LIN {X 0,Y 544.35,Z 282.985,A -85,B 0,C 180,E1 26412.669,E2 26412.669} C_VEL
LIN {X 0,Y 544.407,Z 282.987,A -85,B 0,C 180,E1 26409.453,E2 26409.453} C_VEL
LIN {X 0,Y 544.348,Z 282.987,A -85,B 0,C 180,E1 26406.128,E2 26406.128} C_VEL
LIN {X 0,Y 544.355,Z 282.985,A -85,B 0,C 180,E1 26402.683,E2 26402.683} C_VEL
LIN {X 0,Y 544.403,Z 282.989,A -85,B 0,C 180,E1 26399.482,E2 26399.482} C_VEL
LIN {X 0,Y 544.346,Z 282.986,A -85,B 0,C 180,E1 26396.273,E2 26396.273} C_VEL
LIN {X 0,Y 544.393,Z 282.983,A -85,B 0,C 180,E1 26393.029,E2 26393.029} C_VEL
LIN {X 0,Y 544.372,Z 282.987,A -85,B 0,C 180,E1 26389.751,E2 26389.751} C_VEL
LIN {X 0,Y 544.351,Z 282.985,A -85,B 0,C 180,E1 26386.43,E2 26386.43} C_VEL
LIN {X 0,Y 544.405,Z 282.984,A -85,B 0,C 180,E1 26383.163,E2 26383.163} C_VEL
LIN {X 0,Y 544.358,Z 282.987,A -85,B 0,C 180,E1 26379.941,E2 26379.941} C_VEL
LIN {X 0,Y 544.356,Z 282.984,A -85,B 0,C 180,E1 26376.463,E2 26376.463} C_VEL
LIN {X 0,Y 544.404,Z 282.984,A -85,B 0,C 180,E1 26373.158,E2 26373.158} C_VEL
LIN {X 0,Y 544.36,Z 282.986,A -85,B 0,C 180,E1 26369.894,E2 26369.894} C_VEL
LIN {X 0,Y 544.358,Z 282.984,A -85,B 0,C 180,E1 26366.419,E2 26366.419} C_VEL
LIN {X 0,Y 544.407,Z 282.984,A -85,B 0,C 180,E1 26363.143,E2 26363.143} C_VEL
LIN {X 0,Y 544.363,Z 282.986,A -85,B 0,C 180,E1 26359.843,E2 26359.843} C_VEL
LIN {X 0,Y 544.361,Z 282.984,A -85,B 0,C 180,E1 26356.401,E2 26356.401} C_VEL
LIN {X 0,Y 544.406,Z 282.984,A -85,B 0,C 180,E1 26353.102,E2 26353.102} C_VEL
LIN {X 0,Y 544.366,Z 282.986,A -85,B 0,C 180,E1 26349.799,E2 26349.799} C_VEL
LIN {X 0,Y 544.365,Z 282.983,A -85,B 0,C 180,E1 26346.395,E2 26346.395} C_VEL
LIN {X 0,Y 544.406,Z 282.985,A -85,B 0,C 180,E1 26343.14,E2 26343.14} C_VEL
LIN {X 0,Y 544.362,Z 282.985,A -85,B 0,C 180,E1 26339.89,E2 26339.89} C_VEL
LIN {X 0,Y 544.374,Z 282.982,A -85,B 0,C 180,E1 26336.493,E2 26336.493} C_VEL
LIN {X 0,Y 544.405,Z 282.986,A -85,B 0,C 180,E1 26333.199,E2 26333.199} C_VEL
LIN {X 0,Y 544.361,Z 282.985,A -85,B 0,C 180,E1 26329.986,E2 26329.986} C_VEL
LIN {X 0,Y 544.389,Z 282.981,A -85,B 0,C 180,E1 26326.613,E2 26326.613} C_VEL
LIN {X 0,Y 544.401,Z 282.989,A -85,B 0,C 180,E1 26323.237,E2 26323.237} C_VEL
LIN {X 0,Y 544.364,Z 282.985,A -85,B 0,C 180,E1 26320.002,E2 26320.002} C_VEL
LIN {X 0,Y 544.398,Z 282.982,A -85,B 0,C 180,E1 26316.646,E2 26316.646} C_VEL
LIN {X 0,Y 544.397,Z 282.989,A -85,B 0,C 180,E1 26313.306,E2 26313.306} C_VEL
LIN {X 0,Y 544.365,Z 282.988,A -85,B 0,C 180,E1 26309.971,E2 26309.971} C_VEL
LIN {X 0,Y 544.436,Z 283.218,A -85,B 0,C 180,E1 26308.729,E2 26308.729} C_VEL
LIN {X 0,Y 547.156,Z 294.377,A -85,B 0,C 180,E1 26307.24,E2 26307.24} C_VEL
LIN {X 0,Y 546.527,Z 321.838,A -85,B 0,C 180,E1 26304.018,E2 26304.018} C_VEL
LIN {X 0,Y 545.809,Z 351.894,A -85,B 0,C 180,E1 26300.535,E2 26300.535} C_VEL
LIN {X 0,Y 545.233,Z 382.464,A -85,B 0,C 180,E1 26297.06,E2 26297.06} C_VEL
LIN {X 0,Y 544.899,Z 404.895,A -85,B 0,C 180,E1 26294.573,E2 26294.573} C_VEL
LIN {X 0,Y 545.732,Z 413.339,A -85,B 0,C 180,E1 26294.433,E2 26294.433} C_VEL
LIN {X 0,Y 545.362,Z 516.208,A -85,B 0,C 180,E1 26293.038,E2 26293.038} C_VEL
LIN {X 0,Y 545.216,Z 531.178,A -85,B 0,C 180,E1 26292.642,E2 26292.642} C_VEL
LIN {X 0,Y 544.986,Z 546.217,A -85,B 0,C 180,E1 26292.017,E2 26292.017} C_VEL
LIN {X 0,Y 544.757,Z 559.301,A -85,B 0,C 180,E1 26291.265,E2 26291.265} C_VEL
LIN {X 0,Y 544.54,Z 571.401,A -85,B 0,C 180,E1 26290.365,E2 26290.365} C_VEL
LIN {X 0,Y 544.321,Z 583.569,A -85,B 0,C 180,E1 26289.194,E2 26289.194} C_VEL
LIN {X 0,Y 544.146,Z 593.806,A -85,B 0,C 180,E1 26287.92,E2 26287.92} C_VEL
LIN {X 0,Y 544.035,Z 601.785,A -85,B 0,C 180,E1 26286.647,E2 26286.647} C_VEL
LIN {X 0,Y 543.96,Z 608.864,A -85,B 0,C 180,E1 26285.166,E2 26285.166} C_VEL
LIN {X 0,Y 543.928,Z 614.181,A -85,B 0,C 180,E1 26283.582,E2 26283.582} C_VEL
LIN {X 0,Y 543.917,Z 617.464,A -85,B 0,C 180,E1 26282,E2 26282} C_VEL
LIN {X 0,Y 543.918,Z 618.907,A -85,B 0,C 180,E1 26280.42,E2 26280.42} C_VEL
LIN {X 0,Y 543.915,Z 618.544,A -85,B 0,C 180,E1 26278.84,E2 26278.84} C_VEL
LIN {X 0,Y 543.919,Z 616.339,A -85,B 0,C 180,E1 26277.259,E2 26277.259} C_VEL
LIN {X 0,Y 543.935,Z 612.587,A -85,B 0,C 180,E1 26275.782,E2 26275.782} C_VEL
LIN {X 0,Y 543.983,Z 606.506,A -85,B 0,C 180,E1 26274.197,E2 26274.197} C_VEL
LIN {X 0,Y 544.068,Z 599.221,A -85,B 0,C 180,E1 26272.82,E2 26272.82} C_VEL
LIN {X 0,Y 544.2,Z 590.528,A -85,B 0,C 180,E1 26271.546,E2 26271.546} C_VEL
LIN {X 0,Y 544.389,Z 579.839,A -85,B 0,C 180,E1 26270.324,E2 26270.324} C_VEL
LIN {X 0,Y 544.589,Z 567.853,A -85,B 0,C 180,E1 26269.259,E2 26269.259} C_VEL
LIN {X 0,Y 544.837,Z 555.527,A -85,B 0,C 180,E1 26268.406,E2 26268.406} C_VEL
LIN {X 0,Y 545.075,Z 541.334,A -85,B 0,C 180,E1 26267.659,E2 26267.659} C_VEL
LIN {X 0,Y 545.291,Z 525.913,A -85,B 0,C 180,E1 26267.099,E2 26267.099} C_VEL
LIN {X 0,Y 545.406,Z 510.362,A -85,B 0,C 180,E1 26266.767,E2 26266.767} C_VEL
LIN {X 0,Y 545.638,Z 409.282,A -85,B 0,C 180,E1 26265.372,E2 26265.372} C_VEL
LIN {X 0,Y 544.953,Z 404.69,A -85,B 0,C 180,E1 26265.278,E2 26265.278} C_VEL
LIN {X 0,Y 545.578,Z 374.772,A -85,B 0,C 180,E1 26261.846,E2 26261.846} C_VEL
LIN {X 0,Y 546.318,Z 345.052,A -85,B 0,C 180,E1 26258.394,E2 26258.394} C_VEL
LIN {X 0,Y 547.209,Z 316.527,A -85,B 0,C 180,E1 26255.033,E2 26255.033} C_VEL
LIN {X 0,Y 547.803,Z 295.13,A -85,B 0,C 180,E1 26252.444,E2 26252.444} C_VEL
LIN {X 0,Y 544.407,Z 282.987,A -85,B 0,C 180,E1 26250.634,E2 26250.634} C_VEL
LIN {X 0,Y 544.383,Z 282.99,A -85,B 0,C 180,E1 26247.268,E2 26247.268} C_VEL
LIN {X 0,Y 544.383,Z 282.986,A -85,B 0,C 180,E1 26243.872,E2 26243.872} C_VEL
LIN {X 0,Y 544.393,Z 282.984,A -85,B 0,C 180,E1 26240.544,E2 26240.544} C_VEL
LIN {X 0,Y 544.39,Z 282.988,A -85,B 0,C 180,E1 26237.125,E2 26237.125} C_VEL
LIN {X 0,Y 544.402,Z 282.987,A -85,B 0,C 180,E1 26233.797,E2 26233.797} C_VEL
LIN {X 0,Y 544.387,Z 282.985,A -85,B 0,C 180,E1 26230.418,E2 26230.418} C_VEL
LIN {X 0,Y 544.353,Z 282.99,A -85,B 0,C 180,E1 26227.047,E2 26227.047} C_VEL
LIN {X 0,Y 544.384,Z 282.991,A -85,B 0,C 180,E1 26223.816,E2 26223.816} C_VEL
LIN {X 0,Y 544.345,Z 283.033,A -85,B 0,C 180,E1 26222.92,E2 26222.92} C_VEL
LIN {X 0,Y 549.395,Z 298.474,A -85,B 0,C 180,E1 26221.305,E2 26221.305} C_VEL
LIN {X 0,Y 548.406,Z 338.599,A -85,B 0,C 180,E1 26218.283,E2 26218.283} C_VEL
LIN {X 0,Y 547.611,Z 384.589,A -85,B 0,C 180,E1 26215.005,E2 26215.005} C_VEL
LIN {X 0,Y 547.643,Z 387.567,A -85,B 0,C 180,E1 26214.823,E2 26214.823} C_VEL
LIN {X 0,Y 548.835,Z 396.99,A -85,B 0,C 180,E1 26214.653,E2 26214.653} C_VEL
LIN {X 0,Y 548.051,Z 589.9,A -85,B 0,C 180,E1 26212.072,E2 26212.072} C_VEL
LIN {X 0,Y 547.776,Z 609.321,A -85,B 0,C 180,E1 26211.669,E2 26211.669} C_VEL
LIN {X 0,Y 547.427,Z 627.661,A -85,B 0,C 180,E1 26211.09,E2 26211.09} C_VEL
LIN {X 0,Y 546.99,Z 645.573,A -85,B 0,C 180,E1 26210.323,E2 26210.323} C_VEL
LIN {X 0,Y 546.512,Z 662.304,A -85,B 0,C 180,E1 26209.409,E2 26209.409} C_VEL
LIN {X 0,Y 546.011,Z 678.751,A -85,B 0,C 180,E1 26208.296,E2 26208.296} C_VEL
LIN {X 0,Y 545.512,Z 694.468,A -85,B 0,C 180,E1 26206.999,E2 26206.999} C_VEL
LIN {X 0,Y 545.083,Z 708.249,A -85,B 0,C 180,E1 26205.63,E2 26205.63} C_VEL
LIN {X 0,Y 544.714,Z 720.88,A -85,B 0,C 180,E1 26204.131,E2 26204.131} C_VEL
LIN {X 0,Y 544.42,Z 732.249,A -85,B 0,C 180,E1 26202.517,E2 26202.517} C_VEL
LIN {X 0,Y 544.199,Z 742.233,A -85,B 0,C 180,E1 26200.802,E2 26200.802} C_VEL
LIN {X 0,Y 544.052,Z 750.798,A -85,B 0,C 180,E1 26198.988,E2 26198.988} C_VEL
LIN {X 0,Y 543.974,Z 757.523,A -85,B 0,C 180,E1 26197.181,E2 26197.181} C_VEL
LIN {X 0,Y 543.932,Z 762.857,A -85,B 0,C 180,E1 26195.274,E2 26195.274} C_VEL
LIN {X 0,Y 543.911,Z 766.48,A -85,B 0,C 180,E1 26193.373,E2 26193.373} C_VEL
LIN {X 0,Y 543.912,Z 768.551,A -85,B 0,C 180,E1 26191.37,E2 26191.37} C_VEL
LIN {X 0,Y 543.913,Z 768.872,A -85,B 0,C 180,E1 26189.369,E2 26189.369} C_VEL
LIN {X 0,Y 543.911,Z 767.453,A -85,B 0,C 180,E1 26187.367,E2 26187.367} C_VEL
LIN {X 0,Y 543.92,Z 764.466,A -85,B 0,C 180,E1 26185.467,E2 26185.467} C_VEL
LIN {X 0,Y 543.946,Z 759.811,A -85,B 0,C 180,E1 26183.563,E2 26183.563} C_VEL
LIN {X 0,Y 544.019,Z 753.373,A -85,B 0,C 180,E1 26181.652,E2 26181.652} C_VEL
LIN {X 0,Y 544.141,Z 745.484,A -85,B 0,C 180,E1 26179.841,E2 26179.841} C_VEL
LIN {X 0,Y 544.342,Z 735.601,A -85,B 0,C 180,E1 26178.021,E2 26178.021} C_VEL
LIN {X 0,Y 544.624,Z 724.151,A -85,B 0,C 180,E1 26176.302,E2 26176.302} C_VEL
LIN {X 0,Y 544.998,Z 711.102,A -85,B 0,C 180,E1 26174.682,E2 26174.682} C_VEL
LIN {X 0,Y 545.442,Z 696.892,A -85,B 0,C 180,E1 26173.22,E2 26173.22} C_VEL
LIN {X 0,Y 545.932,Z 681.441,A -85,B 0,C 180,E1 26171.904,E2 26171.904} C_VEL
LIN {X 0,Y 546.426,Z 665.205,A -85,B 0,C 180,E1 26170.768,E2 26170.768} C_VEL
LIN {X 0,Y 546.924,Z 647.857,A -85,B 0,C 180,E1 26169.787,E2 26169.787} C_VEL
LIN {X 0,Y 547.377,Z 629.851,A -85,B 0,C 180,E1 26168.991,E2 26168.991} C_VEL
LIN {X 0,Y 547.749,Z 611.346,A -85,B 0,C 180,E1 26168.385,E2 26168.385} C_VEL
LIN {X 0,Y 548.034,Z 592.5,A -85,B 0,C 180,E1 26167.97,E2 26167.97} C_VEL
LIN {X 0,Y 548.83,Z 394.706,A -85,B 0,C 180,E1 26165.294,E2 26165.294} C_VEL
LIN {X 0,Y 547.652,Z 386.629,A -85,B 0,C 180,E1 26165.114,E2 26165.114} C_VEL
LIN {X 0,Y 548.643,Z 339.725,A -85,B 0,C 180,E1 26161.718,E2 26161.718} C_VEL
LIN {X 0,Y 549.499,Z 299.011,A -85,B 0,C 180,E1 26158.703,E2 26158.703} C_VEL
LIN {X 0,Y 547.135,Z 291.4,A -85,B 0,C 180,E1 26157.988,E2 26157.988} C_VEL
LIN {X 0,Y 544.332,Z 282.995,A -85,B 0,C 180,E1 26157.132,E2 26157.132} C_VEL
LIN {X 0,Y 544.372,Z 282.991,A -85,B 0,C 180,E1 26154.004,E2 26154.004} C_VEL
LIN {X 0,Y 544.32,Z 282.991,A -85,B 0,C 180,E1 26150.811,E2 26150.811} C_VEL
LIN {X 0,Y 544.377,Z 282.99,A -85,B 0,C 180,E1 26147.592,E2 26147.592} C_VEL
LIN {X 0,Y 544.329,Z 282.99,A -85,B 0,C 180,E1 26144.396,E2 26144.396} C_VEL
LIN {X 0,Y 544.325,Z 282.99,A -85,B 0,C 180,E1 26140.979,E2 26140.979} C_VEL
LIN {X 0,Y 544.385,Z 282.989,A -85,B 0,C 180,E1 26137.838,E2 26137.838} C_VEL
LIN {X 0,Y 544.323,Z 282.989,A -85,B 0,C 180,E1 26134.584,E2 26134.584} C_VEL
LIN {X 0,Y 544.354,Z 282.988,A -85,B 0,C 180,E1 26131.32,E2 26131.32} C_VEL
LIN {X 0,Y 544.336,Z 282.989,A -85,B 0,C 180,E1 26128.289,E2 26128.289} C_VEL
LIN {X 0,Y 544.328,Z 282.988,A -85,B 0,C 180,E1 26124.876,E2 26124.876} C_VEL
LIN {X 0,Y 544.396,Z 282.989,A -85,B 0,C 180,E1 26121.665,E2 26121.665} C_VEL
LIN {X 0,Y 544.33,Z 282.988,A -85,B 0,C 180,E1 26118.419,E2 26118.419} C_VEL
LIN {X 0,Y 544.336,Z 282.988,A -85,B 0,C 180,E1 26114.948,E2 26114.948} C_VEL
LIN {X 0,Y 544.386,Z 282.989,A -85,B 0,C 180,E1 26111.765,E2 26111.765} C_VEL
LIN {X 0,Y 544.328,Z 282.988,A -85,B 0,C 180,E1 26108.558,E2 26108.558} C_VEL
LIN {X 0,Y 544.381,Z 282.987,A -85,B 0,C 180,E1 26105.376,E2 26105.376} C_VEL
LIN {X 0,Y 544.341,Z 282.988,A -85,B 0,C 180,E1 26102.212,E2 26102.212} C_VEL
LIN {X 0,Y 544.338,Z 282.987,A -85,B 0,C 180,E1 26098.844,E2 26098.844} C_VEL
LIN {X 0,Y 544.397,Z 282.989,A -85,B 0,C 180,E1 26095.577,E2 26095.577} C_VEL
LIN {X 0,Y 544.333,Z 282.988,A -85,B 0,C 180,E1 26092.402,E2 26092.402} C_VEL
LIN {X 0,Y 544.361,Z 282.986,A -85,B 0,C 180,E1 26089.097,E2 26089.097} C_VEL
LIN {X 0,Y 544.359,Z 282.988,A -85,B 0,C 180,E1 26085.971,E2 26085.971} C_VEL
LIN {X 0,Y 544.339,Z 282.986,A -85,B 0,C 180,E1 26082.69,E2 26082.69} C_VEL
LIN {X 0,Y 544.402,Z 282.987,A -85,B 0,C 180,E1 26079.466,E2 26079.466} C_VEL
LIN {X 0,Y 544.339,Z 282.987,A -85,B 0,C 180,E1 26076.282,E2 26076.282} C_VEL
LIN {X 0,Y 544.355,Z 282.986,A -85,B 0,C 180,E1 26072.904,E2 26072.904} C_VEL
LIN {X 0,Y 544.385,Z 282.989,A -85,B 0,C 180,E1 26069.68,E2 26069.68} C_VEL
LIN {X 0,Y 544.383,Z 282.985,A -85,B 0,C 180,E1 26069.164,E2 26069.164} C_VEL
LIN {X 0,Y 543.331,Z 283.113,A -85,B 0,C 180,E1 26068.354,E2 26068.354} C_VEL
LIN {X 0,Y 536.958,Z 283.922,A -85,B 0,C 180,E1 26066.077,E2 26066.077} C_VEL
LIN {X 0,Y 536.46,Z 283.977,A -85,B 0,C 180,E1 26065.485,E2 26065.485} C_VEL
LIN {X 0,Y 536.406,Z 283.976,A -85,B 0,C 180,E1 26062.178,E2 26062.178} C_VEL
LIN {X 0,Y 536.41,Z 283.974,A -85,B 0,C 180,E1 26058.692,E2 26058.692} C_VEL
LIN {X 0,Y 536.464,Z 283.975,A -85,B 0,C 180,E1 26055.363,E2 26055.363} C_VEL
LIN {X 0,Y 536.41,Z 283.976,A -85,B 0,C 180,E1 26052.113,E2 26052.113} C_VEL
LIN {X 0,Y 536.412,Z 283.974,A -85,B 0,C 180,E1 26048.639,E2 26048.639} C_VEL
LIN {X 0,Y 536.462,Z 283.976,A -85,B 0,C 180,E1 26045.424,E2 26045.424} C_VEL
LIN {X 0,Y 536.408,Z 283.975,A -85,B 0,C 180,E1 26042.199,E2 26042.199} C_VEL
LIN {X 0,Y 536.43,Z 283.973,A -85,B 0,C 180,E1 26038.837,E2 26038.837} C_VEL
LIN {X 0,Y 536.451,Z 283.977,A -85,B 0,C 180,E1 26035.571,E2 26035.571} C_VEL
LIN {X 0,Y 536.41,Z 283.975,A -85,B 0,C 180,E1 26032.233,E2 26032.233} C_VEL
LIN {X 0,Y 536.444,Z 283.972,A -85,B 0,C 180,E1 26028.923,E2 26028.923} C_VEL
LIN {X 0,Y 536.451,Z 283.977,A -85,B 0,C 180,E1 26025.568,E2 26025.568} C_VEL
LIN {X 0,Y 536.411,Z 283.974,A -85,B 0,C 180,E1 26022.268,E2 26022.268} C_VEL
LIN {X 0,Y 536.453,Z 283.972,A -85,B 0,C 180,E1 26018.966,E2 26018.966} C_VEL
LIN {X 0,Y 536.439,Z 283.976,A -85,B 0,C 180,E1 26015.668,E2 26015.668} C_VEL
LIN {X 0,Y 536.416,Z 283.973,A -85,B 0,C 180,E1 26012.349,E2 26012.349} C_VEL
LIN {X 0,Y 536.463,Z 283.972,A -85,B 0,C 180,E1 26009.038,E2 26009.038} C_VEL
LIN {X 0,Y 536.437,Z 283.976,A -85,B 0,C 180,E1 26005.659,E2 26005.659} C_VEL
LIN {X 0,Y 536.417,Z 283.973,A -85,B 0,C 180,E1 26002.287,E2 26002.287} C_VEL
LIN {X 0,Y 536.46,Z 283.971,A -85,B 0,C 180,E1 25998.931,E2 25998.931} C_VEL
LIN {X 0,Y 536.446,Z 283.977,A -85,B 0,C 180,E1 25995.536,E2 25995.536} C_VEL
LIN {X 0,Y 536.419,Z 283.973,A -85,B 0,C 180,E1 25992.2,E2 25992.2} C_VEL
LIN {X 0,Y 536.466,Z 283.97,A -85,B 0,C 180,E1 25988.917,E2 25988.917} C_VEL
LIN {X 0,Y 536.443,Z 283.976,A -85,B 0,C 180,E1 25985.557,E2 25985.557} C_VEL
LIN {X 0,Y 536.423,Z 283.973,A -85,B 0,C 180,E1 25982.225,E2 25982.225} C_VEL
LIN {X 0,Y 536.467,Z 283.971,A -85,B 0,C 180,E1 25978.917,E2 25978.917} C_VEL
LIN {X 0,Y 536.439,Z 283.976,A -85,B 0,C 180,E1 25975.614,E2 25975.614} C_VEL
LIN {X 0,Y 536.425,Z 283.973,A -85,B 0,C 180,E1 25972.176,E2 25972.176} C_VEL
LIN {X 0,Y 536.467,Z 283.97,A -85,B 0,C 180,E1 25968.844,E2 25968.844} C_VEL
LIN {X 0,Y 536.454,Z 283.977,A -85,B 0,C 180,E1 25965.393,E2 25965.393} C_VEL
LIN {X 0,Y 536.425,Z 283.973,A -85,B 0,C 180,E1 25961.998,E2 25961.998} C_VEL
LIN {X 0,Y 536.458,Z 283.971,A -85,B 0,C 180,E1 25958.634,E2 25958.634} C_VEL
LIN {X 0,Y 536.459,Z 283.977,A -85,B 0,C 180,E1 25955.278,E2 25955.278} C_VEL
LIN {X 0,Y 536.425,Z 283.974,A -85,B 0,C 180,E1 25951.959,E2 25951.959} C_VEL
LIN {X 0,Y 536.486,Z 284.117,A -85,B 0,C 180,E1 25949.086,E2 25949.086} C_VEL
LIN {X 0,Y 539.574,Z 296.864,A -85,B 0,C 180,E1 25947.356,E2 25947.356} C_VEL
LIN {X 0,Y 538.85,Z 324.871,A -85,B 0,C 180,E1 25944.033,E2 25944.033} C_VEL
LIN {X 0,Y 538.045,Z 354.443,A -85,B 0,C 180,E1 25940.56,E2 25940.56} C_VEL
LIN {X 0,Y 537.397,Z 384.529,A -85,B 0,C 180,E1 25937.094,E2 25937.094} C_VEL
LIN {X 0,Y 537.089,Z 404.785,A -85,B 0,C 180,E1 25934.837,E2 25934.837} C_VEL
LIN {X 0,Y 538.058,Z 413.957,A -85,B 0,C 180,E1 25934.666,E2 25934.666} C_VEL
LIN {X 0,Y 537.621,Z 515.567,A -85,B 0,C 180,E1 25933.263,E2 25933.263} C_VEL
LIN {X 0,Y 537.452,Z 531.399,A -85,B 0,C 180,E1 25932.847,E2 25932.847} C_VEL
LIN {X 0,Y 537.214,Z 545.837,A -85,B 0,C 180,E1 25932.248,E2 25932.248} C_VEL
LIN {X 0,Y 536.96,Z 559.078,A -85,B 0,C 180,E1 25931.491,E2 25931.491} C_VEL
LIN {X 0,Y 536.7,Z 571.358,A -85,B 0,C 180,E1 25930.572,E2 25930.572} C_VEL
LIN {X 0,Y 536.443,Z 583.028,A -85,B 0,C 180,E1 25929.439,E2 25929.439} C_VEL
LIN {X 0,Y 536.237,Z 592.62,A -85,B 0,C 180,E1 25928.253,E2 25928.253} C_VEL
LIN {X 0,Y 536.075,Z 601.425,A -85,B 0,C 180,E1 25926.854,E2 25926.854} C_VEL
LIN {X 0,Y 535.976,Z 608.485,A -85,B 0,C 180,E1 25925.35,E2 25925.35} C_VEL
LIN {X 0,Y 535.931,Z 613.881,A -85,B 0,C 180,E1 25923.742,E2 25923.742} C_VEL
LIN {X 0,Y 535.918,Z 617.146,A -85,B 0,C 180,E1 25922.244,E2 25922.244} C_VEL
LIN {X 0,Y 535.918,Z 618.828,A -85,B 0,C 180,E1 25920.64,E2 25920.64} C_VEL
LIN {X 0,Y 535.915,Z 618.68,A -85,B 0,C 180,E1 25919.036,E2 25919.036} C_VEL
LIN {X 0,Y 535.919,Z 616.751,A -85,B 0,C 180,E1 25917.432,E2 25917.432} C_VEL
LIN {X 0,Y 535.936,Z 612.913,A -85,B 0,C 180,E1 25915.826,E2 25915.826} C_VEL
LIN {X 0,Y 535.995,Z 607.122,A -85,B 0,C 180,E1 25914.217,E2 25914.217} C_VEL
LIN {X 0,Y 536.106,Z 600.193,A -85,B 0,C 180,E1 25912.82,E2 25912.82} C_VEL
LIN {X 0,Y 536.276,Z 591.881,A -85,B 0,C 180,E1 25911.529,E2 25911.529} C_VEL
LIN {X 0,Y 536.509,Z 581.587,A -85,B 0,C 180,E1 25910.289,E2 25910.289} C_VEL
LIN {X 0,Y 536.747,Z 570.768,A -85,B 0,C 180,E1 25909.263,E2 25909.263} C_VEL
LIN {X 0,Y 537.048,Z 558.043,A -85,B 0,C 180,E1 25908.322,E2 25908.322} C_VEL
LIN {X 0,Y 537.316,Z 543.744,A -85,B 0,C 180,E1 25907.533,E2 25907.533} C_VEL
LIN {X 0,Y 537.53,Z 529.508,A -85,B 0,C 180,E1 25906.978,E2 25906.978} C_VEL
LIN {X 0,Y 537.681,Z 514.748,A -85,B 0,C 180,E1 25906.607,E2 25906.607} C_VEL
LIN {X 0,Y 538.178,Z 410.191,A -85,B 0,C 180,E1 25905.076,E2 25905.076} C_VEL
LIN {X 0,Y 537.255,Z 404.386,A -85,B 0,C 180,E1 25904.924,E2 25904.924} C_VEL
LIN {X 0,Y 537.987,Z 374.156,A -85,B 0,C 180,E1 25901.415,E2 25901.415} C_VEL
LIN {X 0,Y 538.784,Z 344.997,A -85,B 0,C 180,E1 25897.983,E2 25897.983} C_VEL
LIN {X 0,Y 539.793,Z 316.85,A -85,B 0,C 180,E1 25894.607,E2 25894.607} C_VEL
LIN {X 0,Y 540.407,Z 297.828,A -85,B 0,C 180,E1 25892.268,E2 25892.268} C_VEL
LIN {X 0,Y 536.451,Z 283.977,A -85,B 0,C 180,E1 25890.155,E2 25890.155} C_VEL
LIN {X 0,Y 536.463,Z 283.977,A -85,B 0,C 180,E1 25886.772,E2 25886.772} C_VEL
LIN {X 0,Y 536.453,Z 283.978,A -85,B 0,C 180,E1 25883.385,E2 25883.385} C_VEL
LIN {X 0,Y 536.456,Z 283.974,A -85,B 0,C 180,E1 25879.982,E2 25879.982} C_VEL
LIN {X 0,Y 536.446,Z 283.974,A -85,B 0,C 180,E1 25876.628,E2 25876.628} C_VEL
LIN {X 0,Y 536.439,Z 283.978,A -85,B 0,C 180,E1 25873.161,E2 25873.161} C_VEL
LIN {X 0,Y 536.468,Z 283.977,A -85,B 0,C 180,E1 25869.836,E2 25869.836} C_VEL
LIN {X 0,Y 536.436,Z 283.978,A -85,B 0,C 180,E1 25866.484,E2 25866.484} C_VEL
LIN {X 0,Y 536.416,Z 284.026,A -85,B 0,C 180,E1 25863.423,E2 25863.423} C_VEL
LIN {X 0,Y 542.046,Z 300.618,A -85,B 0,C 180,E1 25861.593,E2 25861.593} C_VEL
LIN {X 0,Y 541.211,Z 329.848,A -85,B 0,C 180,E1 25859.308,E2 25859.308} C_VEL
LIN {X 0,Y 540.282,Z 369.736,A -85,B 0,C 180,E1 25856.37,E2 25856.37} C_VEL
LIN {X 0,Y 539.98,Z 387.712,A -85,B 0,C 180,E1 25855.098,E2 25855.098} C_VEL
LIN {X 0,Y 541.236,Z 397.959,A -85,B 0,C 180,E1 25854.906,E2 25854.906} C_VEL
LIN {X 0,Y 540.36,Z 596.253,A -85,B 0,C 180,E1 25852.217,E2 25852.217} C_VEL
LIN {X 0,Y 540.061,Z 615.489,A -85,B 0,C 180,E1 25851.759,E2 25851.759} C_VEL
LIN {X 0,Y 539.684,Z 634.283,A -85,B 0,C 180,E1 25851.109,E2 25851.109} C_VEL
LIN {X 0,Y 539.255,Z 650.939,A -85,B 0,C 180,E1 25850.345,E2 25850.345} C_VEL
LIN {X 0,Y 538.737,Z 666.937,A -85,B 0,C 180,E1 25849.404,E2 25849.404} C_VEL
LIN {X 0,Y 538.177,Z 682.94,A -85,B 0,C 180,E1 25848.244,E2 25848.244} C_VEL
LIN {X 0,Y 537.632,Z 697.935,A -85,B 0,C 180,E1 25846.927,E2 25846.927} C_VEL
LIN {X 0,Y 537.131,Z 712.012,A -85,B 0,C 180,E1 25845.439,E2 25845.439} C_VEL
LIN {X 0,Y 536.711,Z 724.906,A -85,B 0,C 180,E1 25843.796,E2 25843.796} C_VEL
LIN {X 0,Y 536.395,Z 736.223,A -85,B 0,C 180,E1 25842.051,E2 25842.051} C_VEL
LIN {X 0,Y 536.168,Z 745.989,A -85,B 0,C 180,E1 25840.205,E2 25840.205} C_VEL
LIN {X 0,Y 536.024,Z 754.173,A -85,B 0,C 180,E1 25838.259,E2 25838.259} C_VEL
LIN {X 0,Y 535.948,Z 760.41,A -85,B 0,C 180,E1 25836.32,E2 25836.32} C_VEL
LIN {X 0,Y 535.917,Z 764.876,A -85,B 0,C 180,E1 25834.388,E2 25834.388} C_VEL
LIN {X 0,Y 535.912,Z 767.793,A -85,B 0,C 180,E1 25832.353,E2 25832.353} C_VEL
LIN {X 0,Y 535.908,Z 768.939,A -85,B 0,C 180,E1 25830.322,E2 25830.322} C_VEL
LIN {X 0,Y 535.912,Z 768.415,A -85,B 0,C 180,E1 25828.397,E2 25828.397} C_VEL
LIN {X 0,Y 535.913,Z 766.162,A -85,B 0,C 180,E1 25826.364,E2 25826.364} C_VEL
LIN {X 0,Y 535.933,Z 762.353,A -85,B 0,C 180,E1 25824.434,E2 25824.434} C_VEL
LIN {X 0,Y 535.992,Z 756.823,A -85,B 0,C 180,E1 25822.498,E2 25822.498} C_VEL
LIN {X 0,Y 536.102,Z 749.432,A -85,B 0,C 180,E1 25820.554,E2 25820.554} C_VEL
LIN {X 0,Y 536.289,Z 740.523,A -85,B 0,C 180,E1 25818.712,E2 25818.712} C_VEL
LIN {X 0,Y 536.556,Z 730.159,A -85,B 0,C 180,E1 25816.97,E2 25816.97} C_VEL
LIN {X 0,Y 536.917,Z 718.359,A -85,B 0,C 180,E1 25815.33,E2 25815.33} C_VEL
LIN {X 0,Y 537.393,Z 704.694,A -85,B 0,C 180,E1 25813.752,E2 25813.752} C_VEL
LIN {X 0,Y 537.943,Z 689.615,A -85,B 0,C 180,E1 25812.309,E2 25812.309} C_VEL
LIN {X 0,Y 538.521,Z 673.454,A -85,B 0,C 180,E1 25811.04,E2 25811.04} C_VEL
LIN {X 0,Y 539.087,Z 656.677,A -85,B 0,C 180,E1 25809.969,E2 25809.969} C_VEL
LIN {X 0,Y 539.552,Z 640.04,A -85,B 0,C 180,E1 25809.13,E2 25809.13} C_VEL
LIN {X 0,Y 539.966,Z 621.238,A -85,B 0,C 180,E1 25808.411,E2 25808.411} C_VEL
LIN {X 0,Y 540.301,Z 602.396,A -85,B 0,C 180,E1 25807.896,E2 25807.896} C_VEL
LIN {X 0,Y 540.515,Z 581.132,A -85,B 0,C 180,E1 25807.537,E2 25807.537} C_VEL
LIN {X 0,Y 541.221,Z 395.051,A -85,B 0,C 180,E1 25805.002,E2 25805.002} C_VEL
LIN {X 0,Y 540.047,Z 386.903,A -85,B 0,C 180,E1 25804.824,E2 25804.824} C_VEL
LIN {X 0,Y 541.179,Z 340.529,A -85,B 0,C 180,E1 25801.412,E2 25801.412} C_VEL
LIN {X 0,Y 542.136,Z 300.902,A -85,B 0,C 180,E1 25798.438,E2 25798.438} C_VEL
LIN {X 0,Y 536.386,Z 283.985,A -85,B 0,C 180,E1 25796.673,E2 25796.673} C_VEL
LIN {X 0,Y 536.403,Z 283.981,A -85,B 0,C 180,E1 25793.277,E2 25793.277} C_VEL
LIN {X 0,Y 536.417,Z 283.98,A -85,B 0,C 180,E1 25790.12,E2 25790.12} C_VEL
LIN {X 0,Y 536.381,Z 283.98,A -85,B 0,C 180,E1 25786.835,E2 25786.835} C_VEL
LIN {X 0,Y 536.439,Z 283.979,A -85,B 0,C 180,E1 25783.602,E2 25783.602} C_VEL
LIN {X 0,Y 536.395,Z 283.979,A -85,B 0,C 180,E1 25780.326,E2 25780.326} C_VEL
LIN {X 0,Y 536.384,Z 283.978,A -85,B 0,C 180,E1 25776.902,E2 25776.902} C_VEL
LIN {X 0,Y 536.445,Z 283.978,A -85,B 0,C 180,E1 25773.613,E2 25773.613} C_VEL
LIN {X 0,Y 536.387,Z 283.978,A -85,B 0,C 180,E1 25770.467,E2 25770.467} C_VEL
LIN {X 0,Y 536.392,Z 283.977,A -85,B 0,C 180,E1 25767.002,E2 25767.002} C_VEL
LIN {X 0,Y 536.453,Z 283.978,A -85,B 0,C 180,E1 25763.741,E2 25763.741} C_VEL
LIN {X 0,Y 536.39,Z 283.977,A -85,B 0,C 180,E1 25760.515,E2 25760.515} C_VEL
LIN {X 0,Y 536.407,Z 283.977,A -85,B 0,C 180,E1 25757.129,E2 25757.129} C_VEL
LIN {X 0,Y 536.429,Z 283.978,A -85,B 0,C 180,E1 25753.914,E2 25753.914} C_VEL
LIN {X 0,Y 536.389,Z 283.977,A -85,B 0,C 180,E1 25750.636,E2 25750.636} C_VEL
LIN {X 0,Y 536.442,Z 283.976,A -85,B 0,C 180,E1 25747.39,E2 25747.39} C_VEL
LIN {X 0,Y 536.405,Z 283.977,A -85,B 0,C 180,E1 25744.17,E2 25744.17} C_VEL
LIN {X 0,Y 536.395,Z 283.976,A -85,B 0,C 180,E1 25740.749,E2 25740.749} C_VEL
LIN {X 0,Y 536.459,Z 283.977,A -85,B 0,C 180,E1 25737.545,E2 25737.545} C_VEL
LIN {X 0,Y 536.401,Z 283.977,A -85,B 0,C 180,E1 25734.225,E2 25734.225} C_VEL
LIN {X 0,Y 536.4,Z 283.976,A -85,B 0,C 180,E1 25730.777,E2 25730.777} C_VEL
LIN {X 0,Y 536.461,Z 283.976,A -85,B 0,C 180,E1 25727.516,E2 25727.516} C_VEL
LIN {X 0,Y 536.399,Z 283.976,A -85,B 0,C 180,E1 25724.321,E2 25724.321} C_VEL
LIN {X 0,Y 536.411,Z 283.975,A -85,B 0,C 180,E1 25720.912,E2 25720.912} C_VEL
LIN {X 0,Y 536.452,Z 283.978,A -85,B 0,C 180,E1 25717.655,E2 25717.655} C_VEL
LIN {X 0,Y 536.4,Z 283.976,A -85,B 0,C 180,E1 25714.379,E2 25714.379} C_VEL
LIN {X 0,Y 536.426,Z 283.974,A -85,B 0,C 180,E1 25711.015,E2 25711.015} C_VEL
LIN {X 0,Y 536.435,Z 283.977,A -85,B 0,C 180,E1 25707.789,E2 25707.789} C_VEL
LIN {X 0,Y 536.46,Z 283.977,A -85,B 0,C 180,E1 25705.485,E2 25705.485} C_VEL
LIN {X 0,Y 535.479,Z 284.094,A -85,B 0,C 180,E1 25704.662,E2 25704.662} C_VEL
LIN {X 0,Y 528.988,Z 284.901,A -85,B 0,C 180,E1 25702.352,E2 25702.352} C_VEL
LIN {X 0,Y 528.499,Z 284.966,A -85,B 0,C 180,E1 25701.75,E2 25701.75} C_VEL
LIN {X 0,Y 528.466,Z 284.964,A -85,B 0,C 180,E1 25698.391,E2 25698.391} C_VEL
LIN {X 0,Y 528.499,Z 284.962,A -85,B 0,C 180,E1 25695.036,E2 25695.036} C_VEL
LIN {X 0,Y 528.498,Z 284.966,A -85,B 0,C 180,E1 25691.753,E2 25691.753} C_VEL
LIN {X 0,Y 528.468,Z 284.964,A -85,B 0,C 180,E1 25688.442,E2 25688.442} C_VEL
LIN {X 0,Y 528.515,Z 284.961,A -85,B 0,C 180,E1 25685.107,E2 25685.107} C_VEL
LIN {X 0,Y 528.488,Z 284.965,A -85,B 0,C 180,E1 25681.851,E2 25681.851} C_VEL
LIN {X 0,Y 528.472,Z 284.963,A -85,B 0,C 180,E1 25678.474,E2 25678.474} C_VEL
LIN {X 0,Y 528.524,Z 284.962,A -85,B 0,C 180,E1 25675.191,E2 25675.191} C_VEL
LIN {X 0,Y 528.484,Z 284.965,A -85,B 0,C 180,E1 25671.882,E2 25671.882} C_VEL
LIN {X 0,Y 528.474,Z 284.963,A -85,B 0,C 180,E1 25668.418,E2 25668.418} C_VEL
LIN {X 0,Y 528.531,Z 284.96,A -85,B 0,C 180,E1 25665.132,E2 25665.132} C_VEL
LIN {X 0,Y 528.491,Z 284.965,A -85,B 0,C 180,E1 25661.789,E2 25661.789} C_VEL
LIN {X 0,Y 528.474,Z 284.963,A -85,B 0,C 180,E1 25658.376,E2 25658.376} C_VEL
LIN {X 0,Y 528.525,Z 284.961,A -85,B 0,C 180,E1 25655.1,E2 25655.1} C_VEL
LIN {X 0,Y 528.493,Z 284.965,A -85,B 0,C 180,E1 25651.734,E2 25651.734} C_VEL
LIN {X 0,Y 528.478,Z 284.962,A -85,B 0,C 180,E1 25648.373,E2 25648.373} C_VEL
LIN {X 0,Y 528.524,Z 284.96,A -85,B 0,C 180,E1 25645.007,E2 25645.007} C_VEL
LIN {X 0,Y 528.501,Z 284.965,A -85,B 0,C 180,E1 25641.623,E2 25641.623} C_VEL
LIN {X 0,Y 528.478,Z 284.963,A -85,B 0,C 180,E1 25638.209,E2 25638.209} C_VEL
LIN {X 0,Y 528.521,Z 284.959,A -85,B 0,C 180,E1 25634.866,E2 25634.866} C_VEL
LIN {X 0,Y 528.513,Z 284.966,A -85,B 0,C 180,E1 25631.468,E2 25631.468} C_VEL
LIN {X 0,Y 528.48,Z 284.963,A -85,B 0,C 180,E1 25628.116,E2 25628.116} C_VEL
LIN {X 0,Y 528.512,Z 284.959,A -85,B 0,C 180,E1 25624.722,E2 25624.722} C_VEL
LIN {X 0,Y 528.527,Z 284.965,A -85,B 0,C 180,E1 25621.28,E2 25621.28} C_VEL
LIN {X 0,Y 528.486,Z 284.963,A -85,B 0,C 180,E1 25617.883,E2 25617.883} C_VEL
LIN {X 0,Y 528.491,Z 284.961,A -85,B 0,C 180,E1 25614.358,E2 25614.358} C_VEL
LIN {X 0,Y 528.528,Z 284.96,A -85,B 0,C 180,E1 25610.952,E2 25610.952} C_VEL
LIN {X 0,Y 528.503,Z 284.965,A -85,B 0,C 180,E1 25607.543,E2 25607.543} C_VEL
LIN {X 0,Y 528.488,Z 284.961,A -85,B 0,C 180,E1 25604.122,E2 25604.122} C_VEL
LIN {X 0,Y 528.526,Z 284.96,A -85,B 0,C 180,E1 25600.74,E2 25600.74} C_VEL
LIN {X 0,Y 528.514,Z 284.966,A -85,B 0,C 180,E1 25597.385,E2 25597.385} C_VEL
LIN {X 0,Y 528.489,Z 284.964,A -85,B 0,C 180,E1 25594.038,E2 25594.038} C_VEL
LIN {X 0,Y 528.519,Z 284.961,A -85,B 0,C 180,E1 25590.595,E2 25590.595} C_VEL
LIN {X 0,Y 528.51,Z 284.973,A -85,B 0,C 180,E1 25589.462,E2 25589.462} C_VEL
LIN {X 0,Y 531.995,Z 299.249,A -85,B 0,C 180,E1 25587.488,E2 25587.488} C_VEL
LIN {X 0,Y 531.167,Z 327.626,A -85,B 0,C 180,E1 25584.082,E2 25584.082} C_VEL
LIN {X 0,Y 530.295,Z 356.507,A -85,B 0,C 180,E1 25580.643,E2 25580.643} C_VEL
LIN {X 0,Y 529.59,Z 386.156,A -85,B 0,C 180,E1 25577.19,E2 25577.19} C_VEL
LIN {X 0,Y 529.291,Z 404.692,A -85,B 0,C 180,E1 25575.109,E2 25575.109} C_VEL
LIN {X 0,Y 530.427,Z 414.505,A -85,B 0,C 180,E1 25574.919,E2 25574.919} C_VEL
LIN {X 0,Y 529.873,Z 515.888,A -85,B 0,C 180,E1 25573.474,E2 25573.474} C_VEL
LIN {X 0,Y 529.693,Z 531.784,A -85,B 0,C 180,E1 25573.052,E2 25573.052} C_VEL
LIN {X 0,Y 529.452,Z 545.471,A -85,B 0,C 180,E1 25572.485,E2 25572.485} C_VEL
LIN {X 0,Y 529.181,Z 559.027,A -85,B 0,C 180,E1 25571.717,E2 25571.717} C_VEL
LIN {X 0,Y 528.875,Z 572.152,A -85,B 0,C 180,E1 25570.73,E2 25570.73} C_VEL
LIN {X 0,Y 528.594,Z 583.871,A -85,B 0,C 180,E1 25569.58,E2 25569.58} C_VEL
LIN {X 0,Y 528.366,Z 593.512,A -85,B 0,C 180,E1 25568.377,E2 25568.377} C_VEL
LIN {X 0,Y 528.186,Z 602.381,A -85,B 0,C 180,E1 25566.957,E2 25566.957} C_VEL
LIN {X 0,Y 528.072,Z 609.503,A -85,B 0,C 180,E1 25565.431,E2 25565.431} C_VEL
LIN {X 0,Y 528.01,Z 614.576,A -85,B 0,C 180,E1 25563.907,E2 25563.907} C_VEL
LIN {X 0,Y 527.981,Z 617.946,A -85,B 0,C 180,E1 25562.386,E2 25562.386} C_VEL
LIN {X 0,Y 527.975,Z 619.78,A -85,B 0,C 180,E1 25560.649,E2 25560.649} C_VEL
LIN {X 0,Y 527.977,Z 619.661,A -85,B 0,C 180,E1 25559.022,E2 25559.022} C_VEL
LIN {X 0,Y 527.997,Z 617.814,A -85,B 0,C 180,E1 25557.394,E2 25557.394} C_VEL
LIN {X 0,Y 528.044,Z 614.104,A -85,B 0,C 180,E1 25555.764,E2 25555.764} C_VEL
LIN {X 0,Y 528.117,Z 608.766,A -85,B 0,C 180,E1 25554.24,E2 25554.24} C_VEL
LIN {X 0,Y 528.244,Z 601.996,A -85,B 0,C 180,E1 25552.822,E2 25552.822} C_VEL
LIN {X 0,Y 528.449,Z 593.05,A -85,B 0,C 180,E1 25551.402,E2 25551.402} C_VEL
LIN {X 0,Y 528.703,Z 582.918,A -85,B 0,C 180,E1 25550.164,E2 25550.164} C_VEL
LIN {X 0,Y 528.97,Z 571.916,A -85,B 0,C 180,E1 25549.103,E2 25549.103} C_VEL
LIN {X 0,Y 529.285,Z 559.552,A -85,B 0,C 180,E1 25548.171,E2 25548.171} C_VEL
LIN {X 0,Y 529.559,Z 546.084,A -85,B 0,C 180,E1 25547.403,E2 25547.403} C_VEL
LIN {X 0,Y 529.802,Z 532.047,A -85,B 0,C 180,E1 25546.82,E2 25546.82} C_VEL
LIN {X 0,Y 529.978,Z 516.448,A -85,B 0,C 180,E1 25546.4,E2 25546.4} C_VEL
LIN {X 0,Y 530.767,Z 411.203,A -85,B 0,C 180,E1 25544.767,E2 25544.767} C_VEL
LIN {X 0,Y 529.57,Z 404.408,A -85,B 0,C 180,E1 25544.597,E2 25544.597} C_VEL
LIN {X 0,Y 530.417,Z 373.493,A -85,B 0,C 180,E1 25540.966,E2 25540.966} C_VEL
LIN {X 0,Y 531.285,Z 345.323,A -85,B 0,C 180,E1 25537.597,E2 25537.597} C_VEL
LIN {X 0,Y 532.451,Z 316.653,A -85,B 0,C 180,E1 25534.092,E2 25534.092} C_VEL
LIN {X 0,Y 533.049,Z 300.516,A -85,B 0,C 180,E1 25532.065,E2 25532.065} C_VEL
LIN {X 0,Y 529.257,Z 287.498,A -85,B 0,C 180,E1 25530.03,E2 25530.03} C_VEL
LIN {X 0,Y 528.489,Z 284.969,A -85,B 0,C 180,E1 25529.578,E2 25529.578} C_VEL
LIN {X 0,Y 528.517,Z 284.963,A -85,B 0,C 180,E1 25526.152,E2 25526.152} C_VEL
LIN {X 0,Y 528.518,Z 284.965,A -85,B 0,C 180,E1 25522.743,E2 25522.743} C_VEL
LIN {X 0,Y 528.526,Z 284.966,A -85,B 0,C 180,E1 25519.256,E2 25519.256} C_VEL
LIN {X 0,Y 528.523,Z 284.966,A -85,B 0,C 180,E1 25515.726,E2 25515.726} C_VEL
LIN {X 0,Y 528.521,Z 284.963,A -85,B 0,C 180,E1 25512.294,E2 25512.294} C_VEL
LIN {X 0,Y 528.481,Z 284.967,A -85,B 0,C 180,E1 25508.913,E2 25508.913} C_VEL
LIN {X 0,Y 528.487,Z 284.969,A -85,B 0,C 180,E1 25505.509,E2 25505.509} C_VEL
LIN {X 0,Y 528.541,Z 285.135,A -85,B 0,C 180,E1 25503.955,E2 25503.955} C_VEL
LIN {X 0,Y 534.036,Z 301.026,A -85,B 0,C 180,E1 25502.091,E2 25502.091} C_VEL
LIN {X 0,Y 534.859,Z 304.624,A -85,B 0,C 180,E1 25501.725,E2 25501.725} C_VEL
LIN {X 0,Y 533.455,Z 341.59,A -85,B 0,C 180,E1 25498.797,E2 25498.797} C_VEL
LIN {X 0,Y 532.337,Z 384.628,A -85,B 0,C 180,E1 25495.595,E2 25495.595} C_VEL
LIN {X 0,Y 532.359,Z 388.101,A -85,B 0,C 180,E1 25495.377,E2 25495.377} C_VEL
LIN {X 0,Y 533.661,Z 398.888,A -85,B 0,C 180,E1 25495.171,E2 25495.171} C_VEL
LIN {X 0,Y 532.643,Z 595.617,A -85,B 0,C 180,E1 25492.451,E2 25492.451} C_VEL
LIN {X 0,Y 532.308,Z 614.824,A -85,B 0,C 180,E1 25491.987,E2 25491.987} C_VEL
LIN {X 0,Y 531.909,Z 632.85,A -85,B 0,C 180,E1 25491.359,E2 25491.359} C_VEL
LIN {X 0,Y 531.429,Z 650.627,A -85,B 0,C 180,E1 25490.543,E2 25490.543} C_VEL
LIN {X 0,Y 530.894,Z 667.716,A -85,B 0,C 180,E1 25489.552,E2 25489.552} C_VEL
LIN {X 0,Y 530.373,Z 683.811,A -85,B 0,C 180,E1 25488.408,E2 25488.408} C_VEL
LIN {X 0,Y 529.896,Z 697.41,A -85,B 0,C 180,E1 25487.233,E2 25487.233} C_VEL
LIN {X 0,Y 529.35,Z 711.085,A -85,B 0,C 180,E1 25485.784,E2 25485.784} C_VEL
LIN {X 0,Y 528.89,Z 723.363,A -85,B 0,C 180,E1 25484.228,E2 25484.228} C_VEL
LIN {X 0,Y 528.502,Z 734.951,A -85,B 0,C 180,E1 25482.456,E2 25482.456} C_VEL
LIN {X 0,Y 528.246,Z 744.445,A -85,B 0,C 180,E1 25480.691,E2 25480.691} C_VEL
LIN {X 0,Y 528.067,Z 752.553,A -85,B 0,C 180,E1 25478.823,E2 25478.823} C_VEL
LIN {X 0,Y 527.973,Z 759.197,A -85,B 0,C 180,E1 25476.853,E2 25476.853} C_VEL
LIN {X 0,Y 527.933,Z 764.048,A -85,B 0,C 180,E1 25474.89,E2 25474.89} C_VEL
LIN {X 0,Y 527.914,Z 767.224,A -85,B 0,C 180,E1 25472.932,E2 25472.932} C_VEL
LIN {X 0,Y 527.917,Z 768.826,A -85,B 0,C 180,E1 25470.869,E2 25470.869} C_VEL
LIN {X 0,Y 527.914,Z 768.685,A -85,B 0,C 180,E1 25468.807,E2 25468.807} C_VEL
LIN {X 0,Y 527.912,Z 766.798,A -85,B 0,C 180,E1 25466.744,E2 25466.744} C_VEL
LIN {X 0,Y 527.936,Z 763.367,A -85,B 0,C 180,E1 25464.785,E2 25464.785} C_VEL
LIN {X 0,Y 527.987,Z 758.235,A -85,B 0,C 180,E1 25462.821,E2 25462.821} C_VEL
LIN {X 0,Y 528.097,Z 751.262,A -85,B 0,C 180,E1 25460.85,E2 25460.85} C_VEL
LIN {X 0,Y 528.283,Z 742.813,A -85,B 0,C 180,E1 25458.981,E2 25458.981} C_VEL
LIN {X 0,Y 528.568,Z 732.957,A -85,B 0,C 180,E1 25457.214,E2 25457.214} C_VEL
LIN {X 0,Y 528.947,Z 721.736,A -85,B 0,C 180,E1 25455.552,E2 25455.552} C_VEL
LIN {X 0,Y 529.422,Z 709.138,A -85,B 0,C 180,E1 25453.995,E2 25453.995} C_VEL
LIN {X 0,Y 529.958,Z 695.647,A -85,B 0,C 180,E1 25452.601,E2 25452.601} C_VEL
LIN {X 0,Y 530.483,Z 681.018,A -85,B 0,C 180,E1 25451.37,E2 25451.37} C_VEL
LIN {X 0,Y 531.028,Z 664.831,A -85,B 0,C 180,E1 25450.247,E2 25450.247} C_VEL
LIN {X 0,Y 531.563,Z 647.903,A -85,B 0,C 180,E1 25449.292,E2 25449.292} C_VEL
LIN {X 0,Y 532.043,Z 630.243,A -85,B 0,C 180,E1 25448.504,E2 25448.504} C_VEL
LIN {X 0,Y 532.457,Z 611.391,A -85,B 0,C 180,E1 25447.876,E2 25447.876} C_VEL
LIN {X 0,Y 532.785,Z 592.289,A -85,B 0,C 180,E1 25447.45,E2 25447.45} C_VEL
LIN {X 0,Y 533.74,Z 396.083,A -85,B 0,C 180,E1 25444.711,E2 25444.711} C_VEL
LIN {X 0,Y 532.461,Z 386.852,A -85,B 0,C 180,E1 25444.503,E2 25444.503} C_VEL
LIN {X 0,Y 533.731,Z 341.333,A -85,B 0,C 180,E1 25441.099,E2 25441.099} C_VEL
LIN {X 0,Y 534.795,Z 303.618,A -85,B 0,C 180,E1 25438.214,E2 25438.214} C_VEL
LIN {X 0,Y 528.474,Z 284.972,A -85,B 0,C 180,E1 25436.205,E2 25436.205} C_VEL
LIN {X 0,Y 528.445,Z 284.97,A -85,B 0,C 180,E1 25432.875,E2 25432.875} C_VEL
LIN {X 0,Y 528.51,Z 284.967,A -85,B 0,C 180,E1 25429.678,E2 25429.678} C_VEL
LIN {X 0,Y 528.45,Z 284.969,A -85,B 0,C 180,E1 25426.441,E2 25426.441} C_VEL
LIN {X 0,Y 528.446,Z 284.967,A -85,B 0,C 180,E1 25422.934,E2 25422.934} C_VEL
LIN {X 0,Y 528.51,Z 284.967,A -85,B 0,C 180,E1 25419.65,E2 25419.65} C_VEL
LIN {X 0,Y 528.448,Z 284.967,A -85,B 0,C 180,E1 25416.45,E2 25416.45} C_VEL
LIN {X 0,Y 528.454,Z 284.966,A -85,B 0,C 180,E1 25413.019,E2 25413.019} C_VEL
LIN {X 0,Y 528.521,Z 284.967,A -85,B 0,C 180,E1 25409.714,E2 25409.714} C_VEL
LIN {X 0,Y 528.453,Z 284.966,A -85,B 0,C 180,E1 25406.401,E2 25406.401} C_VEL
LIN {X 0,Y 528.454,Z 284.966,A -85,B 0,C 180,E1 25402.941,E2 25402.941} C_VEL
LIN {X 0,Y 528.514,Z 284.968,A -85,B 0,C 180,E1 25399.68,E2 25399.68} C_VEL
LIN {X 0,Y 528.454,Z 284.966,A -85,B 0,C 180,E1 25396.376,E2 25396.376} C_VEL
LIN {X 0,Y 528.455,Z 284.966,A -85,B 0,C 180,E1 25392.902,E2 25392.902} C_VEL
LIN {X 0,Y 528.517,Z 284.966,A -85,B 0,C 180,E1 25389.585,E2 25389.585} C_VEL
LIN {X 0,Y 528.454,Z 284.966,A -85,B 0,C 180,E1 25386.411,E2 25386.411} C_VEL
LIN {X 0,Y 528.462,Z 284.965,A -85,B 0,C 180,E1 25382.93,E2 25382.93} C_VEL
LIN {X 0,Y 528.518,Z 284.967,A -85,B 0,C 180,E1 25379.676,E2 25379.676} C_VEL
LIN {X 0,Y 528.457,Z 284.965,A -85,B 0,C 180,E1 25376.422,E2 25376.422} C_VEL
LIN {X 0,Y 528.476,Z 284.964,A -85,B 0,C 180,E1 25373.047,E2 25373.047} C_VEL
LIN {X 0,Y 528.491,Z 284.966,A -85,B 0,C 180,E1 25369.868,E2 25369.868} C_VEL
LIN {X 0,Y 528.458,Z 284.965,A -85,B 0,C 180,E1 25366.528,E2 25366.528} C_VEL
LIN {X 0,Y 528.507,Z 284.964,A -85,B 0,C 180,E1 25363.29,E2 25363.29} C_VEL
LIN {X 0,Y 528.48,Z 284.966,A -85,B 0,C 180,E1 25359.976,E2 25359.976} C_VEL
LIN {X 0,Y 528.461,Z 284.964,A -85,B 0,C 180,E1 25356.579,E2 25356.579} C_VEL
LIN {X 0,Y 528.509,Z 284.963,A -85,B 0,C 180,E1 25353.242,E2 25353.242} C_VEL
LIN {X 0,Y 528.475,Z 284.965,A -85,B 0,C 180,E1 25350.037,E2 25350.037} C_VEL
LIN {X 0,Y 528.465,Z 284.964,A -85,B 0,C 180,E1 25346.596,E2 25346.596} C_VEL
LIN {X 0,Y 528.52,Z 284.963,A -85,B 0,C 180,E1 25343.29,E2 25343.29} C_VEL
LIN {X 0,Y 528.499,Z 284.966,A -85,B 0,C 180,E1 25341.75,E2 25341.75} C_VEL
LIN {X 0,Y 527.68,Z 285.074,A -85,B 0,C 180,E1 25340.973,E2 25340.973} C_VEL
LIN {X 0,Y 523.615,Z 285.577,A -85,B 0,C 180,E1 25339.577,E2 25339.577} C_VEL
LIN {X 0,Y 520.871,Z 285.91,A -85,B 0,C 180,E1 25338.447,E2 25338.447} C_VEL
LIN {X 0,Y 520.542,Z 285.954,A -85,B 0,C 180,E1 25337.956,E2 25337.956} C_VEL
LIN {X 0,Y 520.53,Z 285.952,A -85,B 0,C 180,E1 25334.515,E2 25334.515} C_VEL
LIN {X 0,Y 520.579,Z 285.951,A -85,B 0,C 180,E1 25331.162,E2 25331.162} C_VEL
LIN {X 0,Y 520.547,Z 285.954,A -85,B 0,C 180,E1 25327.871,E2 25327.871} C_VEL
LIN {X 0,Y 520.532,Z 285.952,A -85,B 0,C 180,E1 25324.513,E2 25324.513} C_VEL
LIN {X 0,Y 520.59,Z 285.95,A -85,B 0,C 180,E1 25321.235,E2 25321.235} C_VEL
LIN {X 0,Y 520.551,Z 285.954,A -85,B 0,C 180,E1 25317.822,E2 25317.822} C_VEL
LIN {X 0,Y 520.533,Z 285.952,A -85,B 0,C 180,E1 25314.391,E2 25314.391} C_VEL
LIN {X 0,Y 520.576,Z 285.95,A -85,B 0,C 180,E1 25311.029,E2 25311.029} C_VEL
LIN {X 0,Y 520.563,Z 285.954,A -85,B 0,C 180,E1 25307.665,E2 25307.665} C_VEL
LIN {X 0,Y 520.534,Z 285.952,A -85,B 0,C 180,E1 25304.346,E2 25304.346} C_VEL
LIN {X 0,Y 520.575,Z 285.95,A -85,B 0,C 180,E1 25300.96,E2 25300.96} C_VEL
LIN {X 0,Y 520.567,Z 285.954,A -85,B 0,C 180,E1 25297.615,E2 25297.615} C_VEL
LIN {X 0,Y 520.535,Z 285.952,A -85,B 0,C 180,E1 25294.295,E2 25294.295} C_VEL
LIN {X 0,Y 520.574,Z 285.949,A -85,B 0,C 180,E1 25290.88,E2 25290.88} C_VEL
LIN {X 0,Y 520.577,Z 285.955,A -85,B 0,C 180,E1 25287.467,E2 25287.467} C_VEL
LIN {X 0,Y 520.54,Z 285.952,A -85,B 0,C 180,E1 25284.046,E2 25284.046} C_VEL
LIN {X 0,Y 520.554,Z 285.95,A -85,B 0,C 180,E1 25280.603,E2 25280.603} C_VEL
LIN {X 0,Y 520.588,Z 285.953,A -85,B 0,C 180,E1 25277.239,E2 25277.239} C_VEL
LIN {X 0,Y 520.544,Z 285.952,A -85,B 0,C 180,E1 25273.942,E2 25273.942} C_VEL
LIN {X 0,Y 520.552,Z 285.95,A -85,B 0,C 180,E1 25270.475,E2 25270.475} C_VEL
LIN {X 0,Y 520.591,Z 285.951,A -85,B 0,C 180,E1 25267.171,E2 25267.171} C_VEL
LIN {X 0,Y 520.552,Z 285.953,A -85,B 0,C 180,E1 25263.76,E2 25263.76} C_VEL
LIN {X 0,Y 520.548,Z 285.95,A -85,B 0,C 180,E1 25260.292,E2 25260.292} C_VEL
LIN {X 0,Y 520.587,Z 285.948,A -85,B 0,C 180,E1 25256.861,E2 25256.861} C_VEL
LIN {X 0,Y 520.577,Z 285.955,A -85,B 0,C 180,E1 25253.398,E2 25253.398} C_VEL
LIN {X 0,Y 520.545,Z 285.951,A -85,B 0,C 180,E1 25250.027,E2 25250.027} C_VEL
LIN {X 0,Y 520.579,Z 285.948,A -85,B 0,C 180,E1 25246.71,E2 25246.71} C_VEL
LIN {X 0,Y 520.582,Z 285.956,A -85,B 0,C 180,E1 25243.285,E2 25243.285} C_VEL
LIN {X 0,Y 520.55,Z 285.953,A -85,B 0,C 180,E1 25239.903,E2 25239.903} C_VEL
LIN {X 0,Y 520.564,Z 285.951,A -85,B 0,C 180,E1 25236.41,E2 25236.41} C_VEL
LIN {X 0,Y 520.589,Z 285.95,A -85,B 0,C 180,E1 25232.931,E2 25232.931} C_VEL
LIN {X 0,Y 520.556,Z 285.964,A -85,B 0,C 180,E1 25229.83,E2 25229.83} C_VEL
LIN {X 0,Y 524.43,Z 301.343,A -85,B 0,C 180,E1 25227.659,E2 25227.659} C_VEL
LIN {X 0,Y 523.499,Z 329.917,A -85,B 0,C 180,E1 25224.189,E2 25224.189} C_VEL
LIN {X 0,Y 522.545,Z 358.572,A -85,B 0,C 180,E1 25220.729,E2 25220.729} C_VEL
LIN {X 0,Y 521.781,Z 388.457,A -85,B 0,C 180,E1 25217.222,E2 25217.222} C_VEL
LIN {X 0,Y 521.5,Z 404.565,A -85,B 0,C 180,E1 25215.39,E2 25215.39} C_VEL
LIN {X 0,Y 522.806,Z 415.312,A -85,B 0,C 180,E1 25215.175,E2 25215.175} C_VEL
LIN {X 0,Y 522.113,Z 517.974,A -85,B 0,C 180,E1 25213.654,E2 25213.654} C_VEL
LIN {X 0,Y 521.927,Z 533.081,A -85,B 0,C 180,E1 25213.232,E2 25213.232} C_VEL
LIN {X 0,Y 521.637,Z 548.458,A -85,B 0,C 180,E1 25212.563,E2 25212.563} C_VEL
LIN {X 0,Y 521.318,Z 562.209,A -85,B 0,C 180,E1 25211.728,E2 25211.728} C_VEL
LIN {X 0,Y 521.02,Z 574.174,A -85,B 0,C 180,E1 25210.782,E2 25210.782} C_VEL
LIN {X 0,Y 520.727,Z 585.733,A -85,B 0,C 180,E1 25209.615,E2 25209.615} C_VEL
LIN {X 0,Y 520.464,Z 595.947,A -85,B 0,C 180,E1 25208.282,E2 25208.282} C_VEL
LIN {X 0,Y 520.283,Z 603.898,A -85,B 0,C 180,E1 25206.952,E2 25206.952} C_VEL
LIN {X 0,Y 520.162,Z 610.959,A -85,B 0,C 180,E1 25205.403,E2 25205.403} C_VEL
LIN {X 0,Y 520.094,Z 616.258,A -85,B 0,C 180,E1 25203.746,E2 25203.746} C_VEL
LIN {X 0,Y 520.061,Z 619.53,A -85,B 0,C 180,E1 25202.092,E2 25202.092} C_VEL
LIN {X 0,Y 520.06,Z 620.991,A -85,B 0,C 180,E1 25200.549,E2 25200.549} C_VEL
LIN {X 0,Y 520.069,Z 620.728,A -85,B 0,C 180,E1 25198.787,E2 25198.787} C_VEL
LIN {X 0,Y 520.1,Z 618.615,A -85,B 0,C 180,E1 25197.133,E2 25197.133} C_VEL
LIN {X 0,Y 520.162,Z 614.985,A -85,B 0,C 180,E1 25195.589,E2 25195.589} C_VEL
LIN {X 0,Y 520.264,Z 609.07,A -85,B 0,C 180,E1 25193.931,E2 25193.931} C_VEL
LIN {X 0,Y 520.437,Z 601.32,A -85,B 0,C 180,E1 25192.381,E2 25192.381} C_VEL
LIN {X 0,Y 520.667,Z 592.576,A -85,B 0,C 180,E1 25191.05,E2 25191.05} C_VEL
LIN {X 0,Y 520.956,Z 582.364,A -85,B 0,C 180,E1 25189.828,E2 25189.828} C_VEL
LIN {X 0,Y 521.285,Z 569.773,A -85,B 0,C 180,E1 25188.66,E2 25188.66} C_VEL
LIN {X 0,Y 521.643,Z 556.353,A -85,B 0,C 180,E1 25187.715,E2 25187.715} C_VEL
LIN {X 0,Y 521.922,Z 542.635,A -85,B 0,C 180,E1 25186.99,E2 25186.99} C_VEL
LIN {X 0,Y 522.172,Z 527.93,A -85,B 0,C 180,E1 25186.44,E2 25186.44} C_VEL
LIN {X 0,Y 522.326,Z 511.958,A -85,B 0,C 180,E1 25186.077,E2 25186.077} C_VEL
LIN {X 0,Y 523.405,Z 412.692,A -85,B 0,C 180,E1 25184.468,E2 25184.468} C_VEL
LIN {X 0,Y 521.899,Z 404.381,A -85,B 0,C 180,E1 25184.256,E2 25184.256} C_VEL
LIN {X 0,Y 522.835,Z 373.866,A -85,B 0,C 180,E1 25180.621,E2 25180.621} C_VEL
LIN {X 0,Y 523.791,Z 346.691,A -85,B 0,C 180,E1 25177.318,E2 25177.318} C_VEL
LIN {X 0,Y 525.125,Z 317.995,A -85,B 0,C 180,E1 25173.742,E2 25173.742} C_VEL
LIN {X 0,Y 525.829,Z 303.697,A -85,B 0,C 180,E1 25171.921,E2 25171.921} C_VEL
LIN {X 0,Y 522.149,Z 291.053,A -85,B 0,C 180,E1 25169.886,E2 25169.886} C_VEL
LIN {X 0,Y 520.577,Z 285.955,A -85,B 0,C 180,E1 25169.019,E2 25169.019} C_VEL
LIN {X 0,Y 520.562,Z 285.956,A -85,B 0,C 180,E1 25165.618,E2 25165.618} C_VEL
LIN {X 0,Y 520.581,Z 285.951,A -85,B 0,C 180,E1 25162.13,E2 25162.13} C_VEL
LIN {X 0,Y 520.574,Z 285.953,A -85,B 0,C 180,E1 25158.645,E2 25158.645} C_VEL
LIN {X 0,Y 520.568,Z 285.956,A -85,B 0,C 180,E1 25155.133,E2 25155.133} C_VEL
LIN {X 0,Y 520.588,Z 285.955,A -85,B 0,C 180,E1 25151.648,E2 25151.648} C_VEL
LIN {X 0,Y 520.586,Z 285.952,A -85,B 0,C 180,E1 25148.204,E2 25148.204} C_VEL
LIN {X 0,Y 520.533,Z 285.961,A -85,B 0,C 180,E1 25144.895,E2 25144.895} C_VEL
LIN {X 0,Y 520.551,Z 285.984,A -85,B 0,C 180,E1 25144.576,E2 25144.576} C_VEL
LIN {X 0,Y 526.218,Z 301.913,A -85,B 0,C 180,E1 25142.574,E2 25142.574} C_VEL
LIN {X 0,Y 527.643,Z 307.304,A -85,B 0,C 180,E1 25141.982,E2 25141.982} C_VEL
LIN {X 0,Y 525.998,Z 343.694,A -85,B 0,C 180,E1 25139.025,E2 25139.025} C_VEL
LIN {X 0,Y 524.652,Z 387.655,A -85,B 0,C 180,E1 25135.68,E2 25135.68} C_VEL
LIN {X 0,Y 526.099,Z 399.902,A -85,B 0,C 180,E1 25135.442,E2 25135.442} C_VEL
LIN {X 0,Y 524.931,Z 594.978,A -85,B 0,C 180,E1 25132.692,E2 25132.692} C_VEL
LIN {X 0,Y 524.562,Z 614.036,A -85,B 0,C 180,E1 25132.225,E2 25132.225} C_VEL
LIN {X 0,Y 524.115,Z 632.398,A -85,B 0,C 180,E1 25131.575,E2 25131.575} C_VEL
LIN {X 0,Y 523.599,Z 650.095,A -85,B 0,C 180,E1 25130.747,E2 25130.747} C_VEL
LIN {X 0,Y 523.013,Z 667.446,A -85,B 0,C 180,E1 25129.721,E2 25129.721} C_VEL
LIN {X 0,Y 522.438,Z 683.869,A -85,B 0,C 180,E1 25128.524,E2 25128.524} C_VEL
LIN {X 0,Y 521.844,Z 699.897,A -85,B 0,C 180,E1 25127.105,E2 25127.105} C_VEL
LIN {X 0,Y 521.312,Z 714.19,A -85,B 0,C 180,E1 25125.577,E2 25125.577} C_VEL
LIN {X 0,Y 520.914,Z 725.597,A -85,B 0,C 180,E1 25124.11,E2 25124.11} C_VEL
LIN {X 0,Y 520.537,Z 736.221,A -85,B 0,C 180,E1 25122.424,E2 25122.424} C_VEL
LIN {X 0,Y 520.25,Z 745.988,A -85,B 0,C 180,E1 25120.521,E2 25120.521} C_VEL
LIN {X 0,Y 520.063,Z 754.172,A -85,B 0,C 180,E1 25118.514,E2 25118.514} C_VEL
LIN {X 0,Y 519.96,Z 760.41,A -85,B 0,C 180,E1 25116.515,E2 25116.515} C_VEL
LIN {X 0,Y 519.923,Z 764.874,A -85,B 0,C 180,E1 25114.523,E2 25114.523} C_VEL
LIN {X 0,Y 519.911,Z 767.791,A -85,B 0,C 180,E1 25112.426,E2 25112.426} C_VEL
LIN {X 0,Y 519.908,Z 768.916,A -85,B 0,C 180,E1 25110.442,E2 25110.442} C_VEL
LIN {X 0,Y 519.911,Z 768.414,A -85,B 0,C 180,E1 25108.348,E2 25108.348} C_VEL
LIN {X 0,Y 519.917,Z 766.16,A -85,B 0,C 180,E1 25106.252,E2 25106.252} C_VEL
LIN {X 0,Y 519.939,Z 762.352,A -85,B 0,C 180,E1 25104.262,E2 25104.262} C_VEL
LIN {X 0,Y 520.018,Z 756.824,A -85,B 0,C 180,E1 25102.266,E2 25102.266} C_VEL
LIN {X 0,Y 520.16,Z 749.43,A -85,B 0,C 180,E1 25100.262,E2 25100.262} C_VEL
LIN {X 0,Y 520.407,Z 740.521,A -85,B 0,C 180,E1 25098.362,E2 25098.362} C_VEL
LIN {X 0,Y 520.757,Z 730.152,A -85,B 0,C 180,E1 25096.567,E2 25096.567} C_VEL
LIN {X 0,Y 521.115,Z 719.753,A -85,B 0,C 180,E1 25095.103,E2 25095.103} C_VEL
LIN {X 0,Y 521.621,Z 706.198,A -85,B 0,C 180,E1 25093.52,E2 25093.52} C_VEL
LIN {X 0,Y 522.182,Z 691.73,A -85,B 0,C 180,E1 25092.11,E2 25092.11} C_VEL
LIN {X 0,Y 522.759,Z 676.342,A -85,B 0,C 180,E1 25090.858,E2 25090.858} C_VEL
LIN {X 0,Y 523.382,Z 659.288,A -85,B 0,C 180,E1 25089.719,E2 25089.719} C_VEL
LIN {X 0,Y 523.953,Z 642.22,A -85,B 0,C 180,E1 25088.801,E2 25088.801} C_VEL
LIN {X 0,Y 524.47,Z 624.575,A -85,B 0,C 180,E1 25088.06,E2 25088.06} C_VEL
LIN {X 0,Y 524.903,Z 606.12,A -85,B 0,C 180,E1 25087.489,E2 25087.489} C_VEL
LIN {X 0,Y 525.206,Z 587.068,A -85,B 0,C 180,E1 25087.105,E2 25087.105} C_VEL
LIN {X 0,Y 526.274,Z 397.077,A -85,B 0,C 180,E1 25084.411,E2 25084.411} C_VEL
LIN {X 0,Y 524.886,Z 387.018,A -85,B 0,C 180,E1 25084.188,E2 25084.188} C_VEL
LIN {X 0,Y 526.276,Z 342.934,A -85,B 0,C 180,E1 25080.837,E2 25080.837} C_VEL
LIN {X 0,Y 527.442,Z 309.096,A -85,B 0,C 180,E1 25078.198,E2 25078.198} C_VEL
LIN {X 0,Y 527.375,Z 306.025,A -85,B 0,C 180,E1 25077.938,E2 25077.938} C_VEL
LIN {X 0,Y 520.574,Z 285.956,A -85,B 0,C 180,E1 25075.754,E2 25075.754} C_VEL
LIN {X 0,Y 520.52,Z 285.959,A -85,B 0,C 180,E1 25072.351,E2 25072.351} C_VEL
LIN {X 0,Y 520.506,Z 285.959,A -85,B 0,C 180,E1 25068.933,E2 25068.933} C_VEL
LIN {X 0,Y 520.56,Z 285.957,A -85,B 0,C 180,E1 25065.604,E2 25065.604} C_VEL
LIN {X 0,Y 520.52,Z 285.956,A -85,B 0,C 180,E1 25062.309,E2 25062.309} C_VEL
LIN {X 0,Y 520.507,Z 285.956,A -85,B 0,C 180,E1 25058.914,E2 25058.914} C_VEL
LIN {X 0,Y 520.566,Z 285.955,A -85,B 0,C 180,E1 25055.591,E2 25055.591} C_VEL
LIN {X 0,Y 520.521,Z 285.956,A -85,B 0,C 180,E1 25052.278,E2 25052.278} C_VEL
LIN {X 0,Y 520.51,Z 285.955,A -85,B 0,C 180,E1 25048.827,E2 25048.827} C_VEL
LIN {X 0,Y 520.56,Z 285.955,A -85,B 0,C 180,E1 25045.481,E2 25045.481} C_VEL
LIN {X 0,Y 520.525,Z 285.955,A -85,B 0,C 180,E1 25042.205,E2 25042.205} C_VEL
LIN {X 0,Y 520.513,Z 285.955,A -85,B 0,C 180,E1 25038.828,E2 25038.828} C_VEL
LIN {X 0,Y 520.569,Z 285.954,A -85,B 0,C 180,E1 25035.486,E2 25035.486} C_VEL
LIN {X 0,Y 520.526,Z 285.955,A -85,B 0,C 180,E1 25032.2,E2 25032.2} C_VEL
LIN {X 0,Y 520.515,Z 285.954,A -85,B 0,C 180,E1 25028.73,E2 25028.73} C_VEL
LIN {X 0,Y 520.576,Z 285.954,A -85,B 0,C 180,E1 25025.512,E2 25025.512} C_VEL
LIN {X 0,Y 520.526,Z 285.955,A -85,B 0,C 180,E1 25022.203,E2 25022.203} C_VEL
LIN {X 0,Y 520.521,Z 285.954,A -85,B 0,C 180,E1 25018.791,E2 25018.791} C_VEL
LIN {X 0,Y 520.573,Z 285.953,A -85,B 0,C 180,E1 25015.427,E2 25015.427} C_VEL
LIN {X 0,Y 520.528,Z 285.955,A -85,B 0,C 180,E1 25012.163,E2 25012.163} C_VEL
LIN {X 0,Y 520.521,Z 285.954,A -85,B 0,C 180,E1 25008.703,E2 25008.703} C_VEL
LIN {X 0,Y 520.584,Z 285.953,A -85,B 0,C 180,E1 25005.429,E2 25005.429} C_VEL
LIN {X 0,Y 520.533,Z 285.954,A -85,B 0,C 180,E1 25002.103,E2 25002.103} C_VEL
LIN {X 0,Y 520.525,Z 285.953,A -85,B 0,C 180,E1 24998.686,E2 24998.686} C_VEL
LIN {X 0,Y 520.581,Z 285.952,A -85,B 0,C 180,E1 24995.371,E2 24995.371} C_VEL
LIN {X 0,Y 520.535,Z 285.954,A -85,B 0,C 180,E1 24992.054,E2 24992.054} C_VEL
LIN {X 0,Y 520.527,Z 285.953,A -85,B 0,C 180,E1 24988.633,E2 24988.633} C_VEL
LIN {X 0,Y 520.577,Z 285.952,A -85,B 0,C 180,E1 24985.288,E2 24985.288} C_VEL
LIN {X 0,Y 520.543,Z 285.954,A -85,B 0,C 180,E1 24981.936,E2 24981.936} C_VEL
LIN {X 0,Y 520.529,Z 285.953,A -85,B 0,C 180,E1 24978.498,E2 24978.498} C_VEL
LIN {X 0,Y 520.542,Z 285.954,A -85,B 0,C 180,E1 24977.956,E2 24977.956} C_VEL
LIN {X 0,Y 519.585,Z 286.078,A -85,B 0,C 180,E1 24977.108,E2 24977.108} C_VEL
LIN {X 0,Y 513.114,Z 286.878,A -85,B 0,C 180,E1 24974.725,E2 24974.725} C_VEL
LIN {X 0,Y 512.594,Z 286.943,A -85,B 0,C 180,E1 24974.103,E2 24974.103} C_VEL
LIN {X 0,Y 512.595,Z 286.941,A -85,B 0,C 180,E1 24970.648,E2 24970.648} C_VEL
LIN {X 0,Y 512.646,Z 286.941,A -85,B 0,C 180,E1 24967.341,E2 24967.341} C_VEL
LIN {X 0,Y 512.606,Z 286.943,A -85,B 0,C 180,E1 24963.906,E2 24963.906} C_VEL
LIN {X 0,Y 512.593,Z 286.941,A -85,B 0,C 180,E1 24960.445,E2 24960.445} C_VEL
LIN {X 0,Y 512.642,Z 286.94,A -85,B 0,C 180,E1 24957.154,E2 24957.154} C_VEL
LIN {X 0,Y 512.623,Z 286.943,A -85,B 0,C 180,E1 24953.69,E2 24953.69} C_VEL
LIN {X 0,Y 512.594,Z 286.941,A -85,B 0,C 180,E1 24950.315,E2 24950.315} C_VEL
LIN {X 0,Y 512.625,Z 286.939,A -85,B 0,C 180,E1 24946.894,E2 24946.894} C_VEL
LIN {X 0,Y 512.636,Z 286.944,A -85,B 0,C 180,E1 24943.535,E2 24943.535} C_VEL
LIN {X 0,Y 512.598,Z 286.942,A -85,B 0,C 180,E1 24940.11,E2 24940.11} C_VEL
LIN {X 0,Y 512.609,Z 286.939,A -85,B 0,C 180,E1 24936.607,E2 24936.607} C_VEL
LIN {X 0,Y 512.648,Z 286.941,A -85,B 0,C 180,E1 24933.242,E2 24933.242} C_VEL
LIN {X 0,Y 512.606,Z 286.942,A -85,B 0,C 180,E1 24929.887,E2 24929.887} C_VEL
LIN {X 0,Y 512.603,Z 286.94,A -85,B 0,C 180,E1 24926.421,E2 24926.421} C_VEL
LIN {X 0,Y 512.652,Z 286.938,A -85,B 0,C 180,E1 24923.054,E2 24923.054} C_VEL
LIN {X 0,Y 512.63,Z 286.943,A -85,B 0,C 180,E1 24919.548,E2 24919.548} C_VEL
LIN {X 0,Y 512.601,Z 286.941,A -85,B 0,C 180,E1 24916.117,E2 24916.117} C_VEL
LIN {X 0,Y 512.631,Z 286.938,A -85,B 0,C 180,E1 24912.754,E2 24912.754} C_VEL
LIN {X 0,Y 512.645,Z 286.944,A -85,B 0,C 180,E1 24909.327,E2 24909.327} C_VEL
LIN {X 0,Y 512.606,Z 286.941,A -85,B 0,C 180,E1 24905.941,E2 24905.941} C_VEL
LIN {X 0,Y 512.617,Z 286.938,A -85,B 0,C 180,E1 24902.466,E2 24902.466} C_VEL
LIN {X 0,Y 512.651,Z 286.94,A -85,B 0,C 180,E1 24899.106,E2 24899.106} C_VEL
LIN {X 0,Y 512.617,Z 286.942,A -85,B 0,C 180,E1 24895.688,E2 24895.688} C_VEL
LIN {X 0,Y 512.609,Z 286.939,A -85,B 0,C 180,E1 24892.178,E2 24892.178} C_VEL
LIN {X 0,Y 512.644,Z 286.937,A -85,B 0,C 180,E1 24888.758,E2 24888.758} C_VEL
LIN {X 0,Y 512.646,Z 286.944,A -85,B 0,C 180,E1 24885.226,E2 24885.226} C_VEL
LIN {X 0,Y 512.611,Z 286.941,A -85,B 0,C 180,E1 24881.831,E2 24881.831} C_VEL
LIN {X 0,Y 512.618,Z 286.94,A -85,B 0,C 180,E1 24878.332,E2 24878.332} C_VEL
LIN {X 0,Y 512.647,Z 286.941,A -85,B 0,C 180,E1 24874.849,E2 24874.849} C_VEL
LIN {X 0,Y 512.641,Z 286.944,A -85,B 0,C 180,E1 24871.319,E2 24871.319} C_VEL
LIN {X 0,Y 512.619,Z 286.949,A -85,B 0,C 180,E1 24870.211,E2 24870.211} C_VEL
LIN {X 0,Y 516.879,Z 303.197,A -85,B 0,C 180,E1 24867.867,E2 24867.867} C_VEL
LIN {X 0,Y 515.855,Z 331.738,A -85,B 0,C 180,E1 24864.358,E2 24864.358} C_VEL
LIN {X 0,Y 514.845,Z 359.99,A -85,B 0,C 180,E1 24860.91,E2 24860.91} C_VEL
LIN {X 0,Y 514.005,Z 389.771,A -85,B 0,C 180,E1 24857.371,E2 24857.371} C_VEL
LIN {X 0,Y 513.732,Z 404.539,A -85,B 0,C 180,E1 24855.677,E2 24855.677} C_VEL
LIN {X 0,Y 515.197,Z 416.003,A -85,B 0,C 180,E1 24855.441,E2 24855.441} C_VEL
LIN {X 0,Y 514.371,Z 519.21,A -85,B 0,C 180,E1 24853.857,E2 24853.857} C_VEL
LIN {X 0,Y 514.174,Z 533.858,A -85,B 0,C 180,E1 24853.435,E2 24853.435} C_VEL
LIN {X 0,Y 513.866,Z 549.204,A -85,B 0,C 180,E1 24852.757,E2 24852.757} C_VEL
LIN {X 0,Y 513.523,Z 562.974,A -85,B 0,C 180,E1 24851.909,E2 24851.909} C_VEL
LIN {X 0,Y 513.201,Z 574.969,A -85,B 0,C 180,E1 24850.948,E2 24850.948} C_VEL
LIN {X 0,Y 512.883,Z 586.583,A -85,B 0,C 180,E1 24849.763,E2 24849.763} C_VEL
LIN {X 0,Y 512.596,Z 596.858,A -85,B 0,C 180,E1 24848.41,E2 24848.41} C_VEL
LIN {X 0,Y 512.395,Z 604.855,A -85,B 0,C 180,E1 24847.06,E2 24847.06} C_VEL
LIN {X 0,Y 512.269,Z 611.537,A -85,B 0,C 180,E1 24845.599,E2 24845.599} C_VEL
LIN {X 0,Y 512.186,Z 616.765,A -85,B 0,C 180,E1 24844.009,E2 24844.009} C_VEL
LIN {X 0,Y 512.15,Z 620.171,A -85,B 0,C 180,E1 24842.46,E2 24842.46} C_VEL
LIN {X 0,Y 512.146,Z 622.094,A -85,B 0,C 180,E1 24840.67,E2 24840.67} C_VEL
LIN {X 0,Y 512.155,Z 622.031,A -85,B 0,C 180,E1 24838.992,E2 24838.992} C_VEL
LIN {X 0,Y 512.19,Z 620.408,A -85,B 0,C 180,E1 24837.425,E2 24837.425} C_VEL
LIN {X 0,Y 512.26,Z 616.807,A -85,B 0,C 180,E1 24835.745,E2 24835.745} C_VEL
LIN {X 0,Y 512.366,Z 611.608,A -85,B 0,C 180,E1 24834.174,E2 24834.174} C_VEL
LIN {X 0,Y 512.531,Z 604.976,A -85,B 0,C 180,E1 24832.714,E2 24832.714} C_VEL
LIN {X 0,Y 512.777,Z 596.147,A -85,B 0,C 180,E1 24831.25,E2 24831.25} C_VEL
LIN {X 0,Y 513.071,Z 586.535,A -85,B 0,C 180,E1 24830.011,E2 24830.011} C_VEL
LIN {X 0,Y 513.411,Z 574.858,A -85,B 0,C 180,E1 24828.825,E2 24828.825} C_VEL
LIN {X 0,Y 513.787,Z 561.856,A -85,B 0,C 180,E1 24827.809,E2 24827.809} C_VEL
LIN {X 0,Y 514.112,Z 548.169,A -85,B 0,C 180,E1 24827,E2 24827} C_VEL
LIN {X 0,Y 514.396,Z 533.916,A -85,B 0,C 180,E1 24826.385,E2 24826.385} C_VEL
LIN {X 0,Y 514.597,Z 518.353,A -85,B 0,C 180,E1 24825.942,E2 24825.942} C_VEL
LIN {X 0,Y 515.946,Z 413.294,A -85,B 0,C 180,E1 24824.138,E2 24824.138} C_VEL
LIN {X 0,Y 514.248,Z 404,A -85,B 0,C 180,E1 24823.856,E2 24823.856} C_VEL
LIN {X 0,Y 515.32,Z 373.375,A -85,B 0,C 180,E1 24820.15,E2 24820.15} C_VEL
LIN {X 0,Y 516.459,Z 345.806,A -85,B 0,C 180,E1 24816.736,E2 24816.736} C_VEL
LIN {X 0,Y 517.919,Z 318.04,A -85,B 0,C 180,E1 24813.205,E2 24813.205} C_VEL
LIN {X 0,Y 518.5,Z 306.382,A -85,B 0,C 180,E1 24811.68,E2 24811.68} C_VEL
LIN {X 0,Y 514.56,Z 292.779,A -85,B 0,C 180,E1 24809.409,E2 24809.409} C_VEL
LIN {X 0,Y 512.647,Z 286.942,A -85,B 0,C 180,E1 24808.304,E2 24808.304} C_VEL
LIN {X 0,Y 512.644,Z 286.943,A -85,B 0,C 180,E1 24804.808,E2 24804.808} C_VEL
LIN {X 0,Y 512.652,Z 286.943,A -85,B 0,C 180,E1 24801.238,E2 24801.238} C_VEL
LIN {X 0,Y 512.642,Z 286.943,A -85,B 0,C 180,E1 24797.709,E2 24797.709} C_VEL
LIN {X 0,Y 512.644,Z 286.941,A -85,B 0,C 180,E1 24794.287,E2 24794.287} C_VEL
LIN {X 0,Y 512.614,Z 286.944,A -85,B 0,C 180,E1 24790.801,E2 24790.801} C_VEL
LIN {X 0,Y 512.604,Z 286.947,A -85,B 0,C 180,E1 24787.266,E2 24787.266} C_VEL
LIN {X 0,Y 512.615,Z 287.096,A -85,B 0,C 180,E1 24785.228,E2 24785.228} C_VEL
LIN {X 0,Y 517.32,Z 299.679,A -85,B 0,C 180,E1 24783.488,E2 24783.488} C_VEL
LIN {X 0,Y 520.515,Z 309.81,A -85,B 0,C 180,E1 24782.278,E2 24782.278} C_VEL
LIN {X 0,Y 518.662,Z 343.569,A -85,B 0,C 180,E1 24779.445,E2 24779.445} C_VEL
LIN {X 0,Y 517.117,Z 385.59,A -85,B 0,C 180,E1 24776.159,E2 24776.159} C_VEL
LIN {X 0,Y 517.123,Z 388.55,A -85,B 0,C 180,E1 24775.968,E2 24775.968} C_VEL
LIN {X 0,Y 518.545,Z 400.86,A -85,B 0,C 180,E1 24775.721,E2 24775.721} C_VEL
LIN {X 0,Y 517.226,Z 594.508,A -85,B 0,C 180,E1 24772.937,E2 24772.937} C_VEL
LIN {X 0,Y 516.822,Z 613.361,A -85,B 0,C 180,E1 24772.468,E2 24772.468} C_VEL
LIN {X 0,Y 516.329,Z 631.946,A -85,B 0,C 180,E1 24771.798,E2 24771.798} C_VEL
LIN {X 0,Y 515.776,Z 649.563,A -85,B 0,C 180,E1 24770.958,E2 24770.958} C_VEL
LIN {X 0,Y 515.15,Z 666.853,A -85,B 0,C 180,E1 24769.916,E2 24769.916} C_VEL
LIN {X 0,Y 514.535,Z 683.224,A -85,B 0,C 180,E1 24768.702,E2 24768.702} C_VEL
LIN {X 0,Y 513.936,Z 698.626,A -85,B 0,C 180,E1 24767.318,E2 24767.318} C_VEL
LIN {X 0,Y 513.388,Z 712.487,A -85,B 0,C 180,E1 24765.823,E2 24765.823} C_VEL
LIN {X 0,Y 512.941,Z 724.939,A -85,B 0,C 180,E1 24764.219,E2 24764.219} C_VEL
LIN {X 0,Y 512.553,Z 736.015,A -85,B 0,C 180,E1 24762.506,E2 24762.506} C_VEL
LIN {X 0,Y 512.278,Z 745.701,A -85,B 0,C 180,E1 24760.686,E2 24760.686} C_VEL
LIN {X 0,Y 512.093,Z 753.341,A -85,B 0,C 180,E1 24758.874,E2 24758.874} C_VEL
LIN {X 0,Y 511.987,Z 759.499,A -85,B 0,C 180,E1 24756.955,E2 24756.955} C_VEL
LIN {X 0,Y 511.935,Z 764.254,A -85,B 0,C 180,E1 24754.931,E2 24754.931} C_VEL
LIN {X 0,Y 511.913,Z 767.336,A -85,B 0,C 180,E1 24752.912,E2 24752.912} C_VEL
LIN {X 0,Y 511.916,Z 768.848,A -85,B 0,C 180,E1 24750.784,E2 24750.784} C_VEL
LIN {X 0,Y 511.914,Z 768.685,A -85,B 0,C 180,E1 24748.77,E2 24748.77} C_VEL
LIN {X 0,Y 511.913,Z 766.956,A -85,B 0,C 180,E1 24746.754,E2 24746.754} C_VEL
LIN {X 0,Y 511.94,Z 763.367,A -85,B 0,C 180,E1 24744.622,E2 24744.622} C_VEL
LIN {X 0,Y 512.007,Z 758.235,A -85,B 0,C 180,E1 24742.596,E2 24742.596} C_VEL
LIN {X 0,Y 512.144,Z 751.665,A -85,B 0,C 180,E1 24740.676,E2 24740.676} C_VEL
LIN {X 0,Y 512.336,Z 743.547,A -85,B 0,C 180,E1 24738.861,E2 24738.861} C_VEL
LIN {X 0,Y 512.653,Z 733.442,A -85,B 0,C 180,E1 24737.04,E2 24737.04} C_VEL
LIN {X 0,Y 513.061,Z 721.922,A -85,B 0,C 180,E1 24735.325,E2 24735.325} C_VEL
LIN {X 0,Y 513.56,Z 708.862,A -85,B 0,C 180,E1 24733.706,E2 24733.706} C_VEL
LIN {X 0,Y 514.174,Z 693.907,A -85,B 0,C 180,E1 24732.166,E2 24732.166} C_VEL
LIN {X 0,Y 514.807,Z 678.39,A -85,B 0,C 180,E1 24730.839,E2 24730.839} C_VEL
LIN {X 0,Y 515.464,Z 661.983,A -85,B 0,C 180,E1 24729.684,E2 24729.684} C_VEL
LIN {X 0,Y 516.108,Z 644.846,A -85,B 0,C 180,E1 24728.707,E2 24728.707} C_VEL
LIN {X 0,Y 516.687,Z 627.312,A -85,B 0,C 180,E1 24727.921,E2 24727.921} C_VEL
LIN {X 0,Y 517.176,Z 608.625,A -85,B 0,C 180,E1 24727.299,E2 24727.299} C_VEL
LIN {X 0,Y 517.55,Z 589.346,A -85,B 0,C 180,E1 24726.874,E2 24726.874} C_VEL
LIN {X 0,Y 518.842,Z 398.208,A -85,B 0,C 180,E1 24724.106,E2 24724.106} C_VEL
LIN {X 0,Y 517.332,Z 387.066,A -85,B 0,C 180,E1 24723.855,E2 24723.855} C_VEL
LIN {X 0,Y 518.846,Z 344.108,A -85,B 0,C 180,E1 24720.534,E2 24720.534} C_VEL
LIN {X 0,Y 520.281,Z 309.331,A -85,B 0,C 180,E1 24717.751,E2 24717.751} C_VEL
LIN {X 0,Y 513.373,Z 289.487,A -85,B 0,C 180,E1 24715.571,E2 24715.571} C_VEL
LIN {X 0,Y 512.588,Z 286.949,A -85,B 0,C 180,E1 24715.28,E2 24715.28} C_VEL
LIN {X 0,Y 512.621,Z 286.946,A -85,B 0,C 180,E1 24711.951,E2 24711.951} C_VEL
LIN {X 0,Y 512.569,Z 286.948,A -85,B 0,C 180,E1 24708.604,E2 24708.604} C_VEL
LIN {X 0,Y 512.574,Z 286.947,A -85,B 0,C 180,E1 24705.08,E2 24705.08} C_VEL
LIN {X 0,Y 512.633,Z 286.945,A -85,B 0,C 180,E1 24701.669,E2 24701.669} C_VEL
LIN {X 0,Y 512.579,Z 286.944,A -85,B 0,C 180,E1 24698.339,E2 24698.339} C_VEL
LIN {X 0,Y 512.569,Z 286.944,A -85,B 0,C 180,E1 24694.859,E2 24694.859} C_VEL
LIN {X 0,Y 512.619,Z 286.944,A -85,B 0,C 180,E1 24691.517,E2 24691.517} C_VEL
LIN {X 0,Y 512.581,Z 286.944,A -85,B 0,C 180,E1 24688.296,E2 24688.296} C_VEL
LIN {X 0,Y 512.572,Z 286.944,A -85,B 0,C 180,E1 24684.798,E2 24684.798} C_VEL
LIN {X 0,Y 512.629,Z 286.943,A -85,B 0,C 180,E1 24681.511,E2 24681.511} C_VEL
LIN {X 0,Y 512.589,Z 286.944,A -85,B 0,C 180,E1 24678.187,E2 24678.187} C_VEL
LIN {X 0,Y 512.576,Z 286.943,A -85,B 0,C 180,E1 24674.807,E2 24674.807} C_VEL
LIN {X 0,Y 512.629,Z 286.943,A -85,B 0,C 180,E1 24671.477,E2 24671.477} C_VEL
LIN {X 0,Y 512.596,Z 286.944,A -85,B 0,C 180,E1 24668.075,E2 24668.075} C_VEL
LIN {X 0,Y 512.576,Z 286.943,A -85,B 0,C 180,E1 24664.701,E2 24664.701} C_VEL
LIN {X 0,Y 512.623,Z 286.942,A -85,B 0,C 180,E1 24661.343,E2 24661.343} C_VEL
LIN {X 0,Y 512.594,Z 286.944,A -85,B 0,C 180,E1 24658.101,E2 24658.101} C_VEL
LIN {X 0,Y 512.579,Z 286.943,A -85,B 0,C 180,E1 24654.629,E2 24654.629} C_VEL
LIN {X 0,Y 512.619,Z 286.942,A -85,B 0,C 180,E1 24651.251,E2 24651.251} C_VEL
LIN {X 0,Y 512.605,Z 286.944,A -85,B 0,C 180,E1 24647.955,E2 24647.955} C_VEL
LIN {X 0,Y 512.582,Z 286.943,A -85,B 0,C 180,E1 24644.618,E2 24644.618} C_VEL
LIN {X 0,Y 512.625,Z 286.941,A -85,B 0,C 180,E1 24641.229,E2 24641.229} C_VEL
LIN {X 0,Y 512.611,Z 286.944,A -85,B 0,C 180,E1 24637.888,E2 24637.888} C_VEL
LIN {X 0,Y 512.584,Z 286.942,A -85,B 0,C 180,E1 24634.466,E2 24634.466} C_VEL
LIN {X 0,Y 512.615,Z 286.941,A -85,B 0,C 180,E1 24631.074,E2 24631.074} C_VEL
LIN {X 0,Y 512.629,Z 286.944,A -85,B 0,C 180,E1 24627.698,E2 24627.698} C_VEL
LIN {X 0,Y 512.586,Z 286.943,A -85,B 0,C 180,E1 24624.325,E2 24624.325} C_VEL
LIN {X 0,Y 512.607,Z 286.941,A -85,B 0,C 180,E1 24620.923,E2 24620.923} C_VEL
LIN {X 0,Y 512.628,Z 286.944,A -85,B 0,C 180,E1 24617.664,E2 24617.664} C_VEL
LIN {X 0,Y 512.59,Z 286.942,A -85,B 0,C 180,E1 24614.289,E2 24614.289} C_VEL
LIN {X 0,Y 512.594,Z 286.943,A -85,B 0,C 180,E1 24614.103,E2 24614.103} C_VEL
LIN {X 0,Y 511.623,Z 287.068,A -85,B 0,C 180,E1 24613.242,E2 24613.242} C_VEL
LIN {X 0,Y 505.174,Z 287.868,A -85,B 0,C 180,E1 24610.822,E2 24610.822} C_VEL
LIN {X 0,Y 504.653,Z 287.931,A -85,B 0,C 180,E1 24610.19,E2 24610.19} C_VEL
LIN {X 0,Y 504.657,Z 287.93,A -85,B 0,C 180,E1 24606.608,E2 24606.608} C_VEL
LIN {X 0,Y 504.701,Z 287.928,A -85,B 0,C 180,E1 24603.145,E2 24603.145} C_VEL
LIN {X 0,Y 504.685,Z 287.932,A -85,B 0,C 180,E1 24599.688,E2 24599.688} C_VEL
LIN {X 0,Y 504.655,Z 287.93,A -85,B 0,C 180,E1 24596.346,E2 24596.346} C_VEL
LIN {X 0,Y 504.682,Z 287.928,A -85,B 0,C 180,E1 24592.899,E2 24592.899} C_VEL
LIN {X 0,Y 504.704,Z 287.933,A -85,B 0,C 180,E1 24589.448,E2 24589.448} C_VEL
LIN {X 0,Y 504.66,Z 287.931,A -85,B 0,C 180,E1 24586.084,E2 24586.084} C_VEL
LIN {X 0,Y 504.661,Z 287.929,A -85,B 0,C 180,E1 24582.471,E2 24582.471} C_VEL
LIN {X 0,Y 504.71,Z 287.928,A -85,B 0,C 180,E1 24579.118,E2 24579.118} C_VEL
LIN {X 0,Y 504.681,Z 287.932,A -85,B 0,C 180,E1 24575.684,E2 24575.684} C_VEL
LIN {X 0,Y 504.66,Z 287.93,A -85,B 0,C 180,E1 24572.27,E2 24572.27} C_VEL
LIN {X 0,Y 504.693,Z 287.927,A -85,B 0,C 180,E1 24568.864,E2 24568.864} C_VEL
LIN {X 0,Y 504.705,Z 287.932,A -85,B 0,C 180,E1 24565.34,E2 24565.34} C_VEL
LIN {X 0,Y 504.667,Z 287.931,A -85,B 0,C 180,E1 24561.913,E2 24561.913} C_VEL
LIN {X 0,Y 504.665,Z 287.929,A -85,B 0,C 180,E1 24558.34,E2 24558.34} C_VEL
LIN {X 0,Y 504.71,Z 287.927,A -85,B 0,C 180,E1 24554.958,E2 24554.958} C_VEL
LIN {X 0,Y 504.702,Z 287.933,A -85,B 0,C 180,E1 24551.399,E2 24551.399} C_VEL
LIN {X 0,Y 504.666,Z 287.93,A -85,B 0,C 180,E1 24547.997,E2 24547.997} C_VEL
LIN {X 0,Y 504.68,Z 287.927,A -85,B 0,C 180,E1 24544.537,E2 24544.537} C_VEL
LIN {X 0,Y 504.714,Z 287.928,A -85,B 0,C 180,E1 24541.093,E2 24541.093} C_VEL
LIN {X 0,Y 504.682,Z 287.931,A -85,B 0,C 180,E1 24537.661,E2 24537.661} C_VEL
LIN {X 0,Y 504.671,Z 287.928,A -85,B 0,C 180,E1 24534.122,E2 24534.122} C_VEL
LIN {X 0,Y 504.698,Z 287.926,A -85,B 0,C 180,E1 24530.657,E2 24530.657} C_VEL
LIN {X 0,Y 504.711,Z 287.93,A -85,B 0,C 180,E1 24527.134,E2 24527.134} C_VEL
LIN {X 0,Y 504.679,Z 287.931,A -85,B 0,C 180,E1 24523.686,E2 24523.686} C_VEL
LIN {X 0,Y 504.676,Z 287.929,A -85,B 0,C 180,E1 24520.228,E2 24520.228} C_VEL
LIN {X 0,Y 504.709,Z 287.929,A -85,B 0,C 180,E1 24516.836,E2 24516.836} C_VEL
LIN {X 0,Y 504.702,Z 287.932,A -85,B 0,C 180,E1 24513.277,E2 24513.277} C_VEL
LIN {X 0,Y 504.717,Z 288.053,A -85,B 0,C 180,E1 24510.579,E2 24510.579} C_VEL
LIN {X 0,Y 509.308,Z 305.852,A -85,B 0,C 180,E1 24507.98,E2 24507.98} C_VEL
LIN {X 0,Y 508.169,Z 334.584,A -85,B 0,C 180,E1 24504.403,E2 24504.403} C_VEL
LIN {X 0,Y 507.11,Z 363.04,A -85,B 0,C 180,E1 24500.906,E2 24500.906} C_VEL
LIN {X 0,Y 506.143,Z 393.522,A -85,B 0,C 180,E1 24497.234,E2 24497.234} C_VEL
LIN {X 0,Y 505.945,Z 404.307,A -85,B 0,C 180,E1 24495.978,E2 24495.978} C_VEL
LIN {X 0,Y 507.593,Z 416.701,A -85,B 0,C 180,E1 24495.713,E2 24495.713} C_VEL
LIN {X 0,Y 506.641,Z 519.881,A -85,B 0,C 180,E1 24494.079,E2 24494.079} C_VEL
LIN {X 0,Y 506.427,Z 534.623,A -85,B 0,C 180,E1 24493.645,E2 24493.645} C_VEL
LIN {X 0,Y 506.1,Z 549.944,A -85,B 0,C 180,E1 24492.956,E2 24492.956} C_VEL
LIN {X 0,Y 505.734,Z 563.735,A -85,B 0,C 180,E1 24492.095,E2 24492.095} C_VEL
LIN {X 0,Y 505.379,Z 576.051,A -85,B 0,C 180,E1 24491.094,E2 24491.094} C_VEL
LIN {X 0,Y 505.042,Z 587.433,A -85,B 0,C 180,E1 24489.916,E2 24489.916} C_VEL
LIN {X 0,Y 504.73,Z 597.769,A -85,B 0,C 180,E1 24488.542,E2 24488.542} C_VEL
LIN {X 0,Y 504.512,Z 605.828,A -85,B 0,C 180,E1 24487.171,E2 24487.171} C_VEL
LIN {X 0,Y 504.359,Z 612.996,A -85,B 0,C 180,E1 24485.573,E2 24485.573} C_VEL
LIN {X 0,Y 504.271,Z 618.41,A -85,B 0,C 180,E1 24483.864,E2 24483.864} C_VEL
LIN {X 0,Y 504.23,Z 621.787,A -85,B 0,C 180,E1 24482.158,E2 24482.158} C_VEL
LIN {X 0,Y 504.229,Z 623.306,A -85,B 0,C 180,E1 24480.566,E2 24480.566} C_VEL
LIN {X 0,Y 504.251,Z 623.106,A -85,B 0,C 180,E1 24478.749,E2 24478.749} C_VEL
LIN {X 0,Y 504.3,Z 621.022,A -85,B 0,C 180,E1 24477.044,E2 24477.044} C_VEL
LIN {X 0,Y 504.39,Z 617.39,A -85,B 0,C 180,E1 24475.451,E2 24475.451} C_VEL
LIN {X 0,Y 504.532,Z 611.461,A -85,B 0,C 180,E1 24473.741,E2 24473.741} C_VEL
LIN {X 0,Y 504.753,Z 603.678,A -85,B 0,C 180,E1 24472.143,E2 24472.143} C_VEL
LIN {X 0,Y 505.034,Z 594.893,A -85,B 0,C 180,E1 24470.771,E2 24470.771} C_VEL
LIN {X 0,Y 505.376,Z 584.644,A -85,B 0,C 180,E1 24469.511,E2 24469.511} C_VEL
LIN {X 0,Y 505.761,Z 572.034,A -85,B 0,C 180,E1 24468.307,E2 24468.307} C_VEL
LIN {X 0,Y 506.17,Z 558.654,A -85,B 0,C 180,E1 24467.333,E2 24467.333} C_VEL
LIN {X 0,Y 506.493,Z 545.139,A -85,B 0,C 180,E1 24466.586,E2 24466.586} C_VEL
LIN {X 0,Y 506.788,Z 530.075,A -85,B 0,C 180,E1 24465.991,E2 24465.991} C_VEL
LIN {X 0,Y 506.983,Z 513.815,A -85,B 0,C 180,E1 24465.594,E2 24465.594} C_VEL
LIN {X 0,Y 508.621,Z 415.013,A -85,B 0,C 180,E1 24463.833,E2 24463.833} C_VEL
LIN {X 0,Y 506.61,Z 404.015,A -85,B 0,C 180,E1 24463.488,E2 24463.488} C_VEL
LIN {X 0,Y 507.779,Z 374.386,A -85,B 0,C 180,E1 24459.842,E2 24459.842} C_VEL
LIN {X 0,Y 509.115,Z 346.443,A -85,B 0,C 180,E1 24456.319,E2 24456.319} C_VEL
LIN {X 0,Y 510.721,Z 319.289,A -85,B 0,C 180,E1 24452.797,E2 24452.797} C_VEL
LIN {X 0,Y 511.326,Z 309.581,A -85,B 0,C 180,E1 24451.501,E2 24451.501} C_VEL
LIN {X 0,Y 507.744,Z 296.998,A -85,B 0,C 180,E1 24449.333,E2 24449.333} C_VEL
LIN {X 0,Y 504.68,Z 287.936,A -85,B 0,C 180,E1 24447.564,E2 24447.564} C_VEL
LIN {X 0,Y 504.699,Z 287.931,A -85,B 0,C 180,E1 24444.097,E2 24444.097} C_VEL
LIN {X 0,Y 504.699,Z 287.931,A -85,B 0,C 180,E1 24440.591,E2 24440.591} C_VEL
LIN {X 0,Y 504.693,Z 287.933,A -85,B 0,C 180,E1 24437.038,E2 24437.038} C_VEL
LIN {X 0,Y 504.705,Z 287.933,A -85,B 0,C 180,E1 24433.524,E2 24433.524} C_VEL
LIN {X 0,Y 504.714,Z 287.932,A -85,B 0,C 180,E1 24429.944,E2 24429.944} C_VEL
LIN {X 0,Y 504.684,Z 287.934,A -85,B 0,C 180,E1 24426.452,E2 24426.452} C_VEL
LIN {X 0,Y 504.718,Z 288.012,A -85,B 0,C 180,E1 24425.972,E2 24425.972} C_VEL
LIN {X 0,Y 509.847,Z 301.652,A -85,B 0,C 180,E1 24423.947,E2 24423.947} C_VEL
LIN {X 0,Y 513.395,Z 312.42,A -85,B 0,C 180,E1 24422.582,E2 24422.582} C_VEL
LIN {X 0,Y 511.381,Z 344.09,A -85,B 0,C 180,E1 24419.842,E2 24419.842} C_VEL
LIN {X 0,Y 509.637,Z 383.913,A -85,B 0,C 180,E1 24416.633,E2 24416.633} C_VEL
LIN {X 0,Y 509.55,Z 388.789,A -85,B 0,C 180,E1 24416.285,E2 24416.285} C_VEL
LIN {X 0,Y 511.025,Z 401.904,A -85,B 0,C 180,E1 24416.014,E2 24416.014} C_VEL
LIN {X 0,Y 509.756,Z 568.089,A -85,B 0,C 180,E1 24413.587,E2 24413.587} C_VEL
LIN {X 0,Y 509.486,Z 596.266,A -85,B 0,C 180,E1 24413.141,E2 24413.141} C_VEL
LIN {X 0,Y 509.022,Z 615.807,A -85,B 0,C 180,E1 24412.617,E2 24412.617} C_VEL
LIN {X 0,Y 508.472,Z 634.286,A -85,B 0,C 180,E1 24411.906,E2 24411.906} C_VEL
LIN {X 0,Y 507.841,Z 652.222,A -85,B 0,C 180,E1 24410.998,E2 24410.998} C_VEL
LIN {X 0,Y 507.182,Z 668.843,A -85,B 0,C 180,E1 24409.942,E2 24409.942} C_VEL
LIN {X 0,Y 506.545,Z 684.711,A -85,B 0,C 180,E1 24408.709,E2 24408.709} C_VEL
LIN {X 0,Y 505.901,Z 700.306,A -85,B 0,C 180,E1 24407.246,E2 24407.246} C_VEL
LIN {X 0,Y 505.315,Z 714.68,A -85,B 0,C 180,E1 24405.612,E2 24405.612} C_VEL
LIN {X 0,Y 504.856,Z 727.369,A -85,B 0,C 180,E1 24403.866,E2 24403.866} C_VEL
LIN {X 0,Y 504.485,Z 738.477,A -85,B 0,C 180,E1 24402.012,E2 24402.012} C_VEL
LIN {X 0,Y 504.244,Z 747.512,A -85,B 0,C 180,E1 24400.165,E2 24400.165} C_VEL
LIN {X 0,Y 504.068,Z 755.214,A -85,B 0,C 180,E1 24398.186,E2 24398.186} C_VEL
LIN {X 0,Y 503.966,Z 761.221,A -85,B 0,C 180,E1 24396.151,E2 24396.151} C_VEL
LIN {X 0,Y 503.924,Z 765.47,A -85,B 0,C 180,E1 24394.097,E2 24394.097} C_VEL
LIN {X 0,Y 503.914,Z 767.981,A -85,B 0,C 180,E1 24392.048,E2 24392.048} C_VEL
LIN {X 0,Y 503.918,Z 768.815,A -85,B 0,C 180,E1 24390.001,E2 24390.001} C_VEL
LIN {X 0,Y 503.915,Z 767.896,A -85,B 0,C 180,E1 24387.84,E2 24387.84} C_VEL
LIN {X 0,Y 503.923,Z 765.308,A -85,B 0,C 180,E1 24385.791,E2 24385.791} C_VEL
LIN {X 0,Y 503.968,Z 760.921,A -85,B 0,C 180,E1 24383.708,E2 24383.708} C_VEL
LIN {X 0,Y 504.074,Z 754.837,A -85,B 0,C 180,E1 24381.675,E2 24381.675} C_VEL
LIN {X 0,Y 504.246,Z 747.18,A -85,B 0,C 180,E1 24379.721,E2 24379.721} C_VEL
LIN {X 0,Y 504.512,Z 737.511,A -85,B 0,C 180,E1 24377.758,E2 24377.758} C_VEL
LIN {X 0,Y 504.906,Z 726.249,A -85,B 0,C 180,E1 24375.903,E2 24375.903} C_VEL
LIN {X 0,Y 505.404,Z 713.399,A -85,B 0,C 180,E1 24374.158,E2 24374.158} C_VEL
LIN {X 0,Y 506.012,Z 699.457,A -85,B 0,C 180,E1 24372.582,E2 24372.582} C_VEL
LIN {X 0,Y 506.667,Z 684.56,A -85,B 0,C 180,E1 24371.178,E2 24371.178} C_VEL
LIN {X 0,Y 507.35,Z 668.825,A -85,B 0,C 180,E1 24369.947,E2 24369.947} C_VEL
LIN {X 0,Y 508.052,Z 652.216,A -85,B 0,C 180,E1 24368.884,E2 24368.884} C_VEL
LIN {X 0,Y 508.725,Z 634.565,A -85,B 0,C 180,E1 24367.983,E2 24367.983} C_VEL
LIN {X 0,Y 509.338,Z 615.521,A -85,B 0,C 180,E1 24367.247,E2 24367.247} C_VEL
LIN {X 0,Y 509.823,Z 596.51,A -85,B 0,C 180,E1 24366.736,E2 24366.736} C_VEL
LIN {X 0,Y 510.15,Z 565.771,A -85,B 0,C 180,E1 24366.245,E2 24366.245} C_VEL
LIN {X 0,Y 511.395,Z 399.168,A -85,B 0,C 180,E1 24363.787,E2 24363.787} C_VEL
LIN {X 0,Y 509.801,Z 386.978,A -85,B 0,C 180,E1 24363.502,E2 24363.502} C_VEL
LIN {X 0,Y 511.451,Z 344.744,A -85,B 0,C 180,E1 24360.181,E2 24360.181} C_VEL
LIN {X 0,Y 512.963,Z 311.994,A -85,B 0,C 180,E1 24357.496,E2 24357.496} C_VEL
LIN {X 0,Y 505.652,Z 290.951,A -85,B 0,C 180,E1 24355.147,E2 24355.147} C_VEL
LIN {X 0,Y 504.631,Z 287.94,A -85,B 0,C 180,E1 24354.791,E2 24354.791} C_VEL
LIN {X 0,Y 504.65,Z 287.937,A -85,B 0,C 180,E1 24351.319,E2 24351.319} C_VEL
LIN {X 0,Y 504.676,Z 287.935,A -85,B 0,C 180,E1 24347.962,E2 24347.962} C_VEL
LIN {X 0,Y 504.628,Z 287.936,A -85,B 0,C 180,E1 24344.66,E2 24344.66} C_VEL
LIN {X 0,Y 504.639,Z 287.935,A -85,B 0,C 180,E1 24341.134,E2 24341.134} C_VEL
LIN {X 0,Y 504.695,Z 287.934,A -85,B 0,C 180,E1 24337.747,E2 24337.747} C_VEL
LIN {X 0,Y 504.644,Z 287.933,A -85,B 0,C 180,E1 24334.291,E2 24334.291} C_VEL
LIN {X 0,Y 504.632,Z 287.933,A -85,B 0,C 180,E1 24330.877,E2 24330.877} C_VEL
LIN {X 0,Y 504.692,Z 287.933,A -85,B 0,C 180,E1 24327.62,E2 24327.62} C_VEL
LIN {X 0,Y 504.648,Z 287.933,A -85,B 0,C 180,E1 24324.214,E2 24324.214} C_VEL
LIN {X 0,Y 504.633,Z 287.933,A -85,B 0,C 180,E1 24320.743,E2 24320.743} C_VEL
LIN {X 0,Y 504.679,Z 287.932,A -85,B 0,C 180,E1 24317.408,E2 24317.408} C_VEL
LIN {X 0,Y 504.654,Z 287.933,A -85,B 0,C 180,E1 24314.106,E2 24314.106} C_VEL
LIN {X 0,Y 504.636,Z 287.932,A -85,B 0,C 180,E1 24310.665,E2 24310.665} C_VEL
LIN {X 0,Y 504.673,Z 287.932,A -85,B 0,C 180,E1 24307.286,E2 24307.286} C_VEL
LIN {X 0,Y 504.665,Z 287.933,A -85,B 0,C 180,E1 24303.978,E2 24303.978} C_VEL
LIN {X 0,Y 504.637,Z 287.932,A -85,B 0,C 180,E1 24300.569,E2 24300.569} C_VEL
LIN {X 0,Y 504.667,Z 287.931,A -85,B 0,C 180,E1 24297.163,E2 24297.163} C_VEL
LIN {X 0,Y 504.688,Z 287.933,A -85,B 0,C 180,E1 24293.746,E2 24293.746} C_VEL
LIN {X 0,Y 504.641,Z 287.932,A -85,B 0,C 180,E1 24290.421,E2 24290.421} C_VEL
LIN {X 0,Y 504.656,Z 287.931,A -85,B 0,C 180,E1 24286.948,E2 24286.948} C_VEL
LIN {X 0,Y 504.705,Z 287.933,A -85,B 0,C 180,E1 24283.545,E2 24283.545} C_VEL
LIN {X 0,Y 504.658,Z 287.932,A -85,B 0,C 180,E1 24280.078,E2 24280.078} C_VEL
LIN {X 0,Y 504.648,Z 287.931,A -85,B 0,C 180,E1 24276.658,E2 24276.658} C_VEL
LIN {X 0,Y 504.695,Z 287.93,A -85,B 0,C 180,E1 24273.277,E2 24273.277} C_VEL
LIN {X 0,Y 504.668,Z 287.932,A -85,B 0,C 180,E1 24269.92,E2 24269.92} C_VEL
LIN {X 0,Y 504.648,Z 287.931,A -85,B 0,C 180,E1 24266.523,E2 24266.523} C_VEL
LIN {X 0,Y 504.684,Z 287.93,A -85,B 0,C 180,E1 24263.112,E2 24263.112} C_VEL
LIN {X 0,Y 504.68,Z 287.932,A -85,B 0,C 180,E1 24259.773,E2 24259.773} C_VEL
LIN {X 0,Y 504.649,Z 287.931,A -85,B 0,C 180,E1 24256.414,E2 24256.414} C_VEL
LIN {X 0,Y 504.677,Z 287.929,A -85,B 0,C 180,E1 24252.962,E2 24252.962} C_VEL
LIN {X 0,Y 504.653,Z 287.931,A -85,B 0,C 180,E1 24250.19,E2 24250.19} C_VEL
LIN {X 0,Y 503.68,Z 288.058,A -85,B 0,C 180,E1 24249.316,E2 24249.316} C_VEL
LIN {X 0,Y 497.144,Z 288.868,A -85,B 0,C 180,E1 24246.793,E2 24246.793} C_VEL
LIN {X 0,Y 496.715,Z 288.92,A -85,B 0,C 180,E1 24246.215,E2 24246.215} C_VEL
LIN {X 0,Y 496.722,Z 288.918,A -85,B 0,C 180,E1 24242.646,E2 24242.646} C_VEL
LIN {X 0,Y 496.773,Z 288.918,A -85,B 0,C 180,E1 24239.279,E2 24239.279} C_VEL
LIN {X 0,Y 496.731,Z 288.92,A -85,B 0,C 180,E1 24235.88,E2 24235.88} C_VEL
LIN {X 0,Y 496.718,Z 288.919,A -85,B 0,C 180,E1 24232.36,E2 24232.36} C_VEL
LIN {X 0,Y 496.748,Z 288.917,A -85,B 0,C 180,E1 24228.908,E2 24228.908} C_VEL
LIN {X 0,Y 496.769,Z 288.921,A -85,B 0,C 180,E1 24225.406,E2 24225.406} C_VEL
LIN {X 0,Y 496.725,Z 288.92,A -85,B 0,C 180,E1 24221.965,E2 24221.965} C_VEL
LIN {X 0,Y 496.722,Z 288.918,A -85,B 0,C 180,E1 24218.449,E2 24218.449} C_VEL
LIN {X 0,Y 496.767,Z 288.917,A -85,B 0,C 180,E1 24215.08,E2 24215.08} C_VEL
LIN {X 0,Y 496.747,Z 288.921,A -85,B 0,C 180,E1 24211.614,E2 24211.614} C_VEL
LIN {X 0,Y 496.722,Z 288.919,A -85,B 0,C 180,E1 24208.154,E2 24208.154} C_VEL
LIN {X 0,Y 496.742,Z 288.917,A -85,B 0,C 180,E1 24204.687,E2 24204.687} C_VEL
LIN {X 0,Y 496.773,Z 288.918,A -85,B 0,C 180,E1 24201.185,E2 24201.185} C_VEL
LIN {X 0,Y 496.742,Z 288.92,A -85,B 0,C 180,E1 24197.68,E2 24197.68} C_VEL
LIN {X 0,Y 496.726,Z 288.918,A -85,B 0,C 180,E1 24194.178,E2 24194.178} C_VEL
LIN {X 0,Y 496.753,Z 288.916,A -85,B 0,C 180,E1 24190.724,E2 24190.724} C_VEL
LIN {X 0,Y 496.776,Z 288.918,A -85,B 0,C 180,E1 24187.185,E2 24187.185} C_VEL
LIN {X 0,Y 496.739,Z 288.92,A -85,B 0,C 180,E1 24183.715,E2 24183.715} C_VEL
LIN {X 0,Y 496.729,Z 288.918,A -85,B 0,C 180,E1 24180.17,E2 24180.17} C_VEL
LIN {X 0,Y 496.754,Z 288.915,A -85,B 0,C 180,E1 24176.667,E2 24176.667} C_VEL
LIN {X 0,Y 496.772,Z 288.919,A -85,B 0,C 180,E1 24173.144,E2 24173.144} C_VEL
LIN {X 0,Y 496.738,Z 288.92,A -85,B 0,C 180,E1 24169.714,E2 24169.714} C_VEL
LIN {X 0,Y 496.733,Z 288.917,A -85,B 0,C 180,E1 24166.176,E2 24166.176} C_VEL
LIN {X 0,Y 496.763,Z 288.915,A -85,B 0,C 180,E1 24162.707,E2 24162.707} C_VEL
LIN {X 0,Y 496.774,Z 288.921,A -85,B 0,C 180,E1 24159.194,E2 24159.194} C_VEL
LIN {X 0,Y 496.739,Z 288.922,A -85,B 0,C 180,E1 24155.71,E2 24155.71} C_VEL
LIN {X 0,Y 496.739,Z 288.917,A -85,B 0,C 180,E1 24152.233,E2 24152.233} C_VEL
LIN {X 0,Y 496.791,Z 289.049,A -85,B 0,C 180,E1 24150.975,E2 24150.975} C_VEL
LIN {X 0,Y 501.732,Z 307.857,A -85,B 0,C 180,E1 24148.181,E2 24148.181} C_VEL
LIN {X 0,Y 500.556,Z 335.847,A -85,B 0,C 180,E1 24144.65,E2 24144.65} C_VEL
LIN {X 0,Y 499.429,Z 364.476,A -85,B 0,C 180,E1 24141.101,E2 24141.101} C_VEL
LIN {X 0,Y 498.369,Z 394.812,A -85,B 0,C 180,E1 24137.391,E2 24137.391} C_VEL
LIN {X 0,Y 498.176,Z 404.197,A -85,B 0,C 180,E1 24136.286,E2 24136.286} C_VEL
LIN {X 0,Y 499.993,Z 417.433,A -85,B 0,C 180,E1 24135.99,E2 24135.99} C_VEL
LIN {X 0,Y 498.919,Z 520.489,A -85,B 0,C 180,E1 24134.309,E2 24134.309} C_VEL
LIN {X 0,Y 498.686,Z 535.359,A -85,B 0,C 180,E1 24133.861,E2 24133.861} C_VEL
LIN {X 0,Y 498.338,Z 550.66,A -85,B 0,C 180,E1 24133.161,E2 24133.161} C_VEL
LIN {X 0,Y 497.947,Z 564.47,A -85,B 0,C 180,E1 24132.287,E2 24132.287} C_VEL
LIN {X 0,Y 497.575,Z 576.558,A -85,B 0,C 180,E1 24131.296,E2 24131.296} C_VEL
LIN {X 0,Y 497.203,Z 588.269,A -85,B 0,C 180,E1 24130.074,E2 24130.074} C_VEL
LIN {X 0,Y 496.866,Z 598.664,A -85,B 0,C 180,E1 24128.679,E2 24128.679} C_VEL
LIN {X 0,Y 496.627,Z 606.782,A -85,B 0,C 180,E1 24127.285,E2 24127.285} C_VEL
LIN {X 0,Y 496.469,Z 613.568,A -85,B 0,C 180,E1 24125.778,E2 24125.778} C_VEL
LIN {X 0,Y 496.365,Z 618.849,A -85,B 0,C 180,E1 24124.157,E2 24124.157} C_VEL
LIN {X 0,Y 496.319,Z 622.396,A -85,B 0,C 180,E1 24122.538,E2 24122.538} C_VEL
LIN {X 0,Y 496.315,Z 624.409,A -85,B 0,C 180,E1 24120.691,E2 24120.691} C_VEL
LIN {X 0,Y 496.334,Z 624.401,A -85,B 0,C 180,E1 24118.96,E2 24118.96} C_VEL
LIN {X 0,Y 496.386,Z 622.805,A -85,B 0,C 180,E1 24117.343,E2 24117.343} C_VEL
LIN {X 0,Y 496.485,Z 619.214,A -85,B 0,C 180,E1 24115.609,E2 24115.609} C_VEL
LIN {X 0,Y 496.626,Z 613.998,A -85,B 0,C 180,E1 24113.989,E2 24113.989} C_VEL
LIN {X 0,Y 496.835,Z 607.337,A -85,B 0,C 180,E1 24112.482,E2 24112.482} C_VEL
LIN {X 0,Y 497.146,Z 598.22,A -85,B 0,C 180,E1 24110.934,E2 24110.934} C_VEL
LIN {X 0,Y 497.507,Z 588.17,A -85,B 0,C 180,E1 24109.617,E2 24109.617} C_VEL
LIN {X 0,Y 497.886,Z 577.162,A -85,B 0,C 180,E1 24108.472,E2 24108.472} C_VEL
LIN {X 0,Y 498.308,Z 564.482,A -85,B 0,C 180,E1 24107.445,E2 24107.445} C_VEL
LIN {X 0,Y 498.684,Z 551.038,A -85,B 0,C 180,E1 24106.609,E2 24106.609} C_VEL
LIN {X 0,Y 499.027,Z 536.421,A -85,B 0,C 180,E1 24105.939,E2 24105.939} C_VEL
LIN {X 0,Y 499.28,Z 520.324,A -85,B 0,C 180,E1 24105.45,E2 24105.45} C_VEL
LIN {X 0,Y 501.186,Z 415.732,A -85,B 0,C 180,E1 24103.471,E2 24103.471} C_VEL
LIN {X 0,Y 499.011,Z 404.111,A -85,B 0,C 180,E1 24103.109,E2 24103.109} C_VEL
LIN {X 0,Y 500.31,Z 374.555,A -85,B 0,C 180,E1 24099.405,E2 24099.405} C_VEL
LIN {X 0,Y 501.843,Z 346.912,A -85,B 0,C 180,E1 24095.856,E2 24095.856} C_VEL
LIN {X 0,Y 503.634,Z 320.15,A -85,B 0,C 180,E1 24092.307,E2 24092.307} C_VEL
LIN {X 0,Y 504.107,Z 312.475,A -85,B 0,C 180,E1 24091.245,E2 24091.245} C_VEL
LIN {X 0,Y 500.797,Z 300.708,A -85,B 0,C 180,E1 24089.151,E2 24089.151} C_VEL
LIN {X 0,Y 497.637,Z 291.717,A -85,B 0,C 180,E1 24087.338,E2 24087.338} C_VEL
LIN {X 0,Y 496.769,Z 288.922,A -85,B 0,C 180,E1 24086.737,E2 24086.737} C_VEL
LIN {X 0,Y 496.767,Z 288.922,A -85,B 0,C 180,E1 24083.144,E2 24083.144} C_VEL
LIN {X 0,Y 496.762,Z 288.922,A -85,B 0,C 180,E1 24079.6,E2 24079.6} C_VEL
LIN {X 0,Y 496.769,Z 288.919,A -85,B 0,C 180,E1 24076.02,E2 24076.02} C_VEL
LIN {X 0,Y 496.751,Z 288.921,A -85,B 0,C 180,E1 24072.549,E2 24072.549} C_VEL
LIN {X 0,Y 496.728,Z 288.925,A -85,B 0,C 180,E1 24069.015,E2 24069.015} C_VEL
LIN {X 0,Y 496.74,Z 289.032,A -85,B 0,C 180,E1 24066.819,E2 24066.819} C_VEL
LIN {X 0,Y 498.127,Z 292.488,A -85,B 0,C 180,E1 24066.204,E2 24066.204} C_VEL
LIN {X 0,Y 502.643,Z 304.202,A -85,B 0,C 180,E1 24064.358,E2 24064.358} C_VEL
LIN {X 0,Y 506.292,Z 315.41,A -85,B 0,C 180,E1 24062.861,E2 24062.861} C_VEL
LIN {X 0,Y 504.025,Z 346.978,A -85,B 0,C 180,E1 24060.06,E2 24060.06} C_VEL
LIN {X 0,Y 502.024,Z 387.07,A -85,B 0,C 180,E1 24056.752,E2 24056.752} C_VEL
LIN {X 0,Y 502.05,Z 389.286,A -85,B 0,C 180,E1 24056.616,E2 24056.616} C_VEL
LIN {X 0,Y 503.554,Z 402.911,A -85,B 0,C 180,E1 24056.326,E2 24056.326} C_VEL
LIN {X 0,Y 502.193,Z 553.177,A -85,B 0,C 180,E1 24054.062,E2 24054.062} C_VEL
LIN {X 0,Y 501.839,Z 593.91,A -85,B 0,C 180,E1 24053.442,E2 24053.442} C_VEL
LIN {X 0,Y 501.353,Z 612.838,A -85,B 0,C 180,E1 24052.948,E2 24052.948} C_VEL
LIN {X 0,Y 500.765,Z 631.749,A -85,B 0,C 180,E1 24052.233,E2 24052.233} C_VEL
LIN {X 0,Y 500.11,Z 649.583,A -85,B 0,C 180,E1 24051.339,E2 24051.339} C_VEL
LIN {X 0,Y 499.402,Z 666.547,A -85,B 0,C 180,E1 24050.266,E2 24050.266} C_VEL
LIN {X 0,Y 498.708,Z 682.664,A -85,B 0,C 180,E1 24049.015,E2 24049.015} C_VEL
LIN {X 0,Y 498.049,Z 697.864,A -85,B 0,C 180,E1 24047.587,E2 24047.587} C_VEL
LIN {X 0,Y 497.434,Z 712.042,A -85,B 0,C 180,E1 24045.985,E2 24045.985} C_VEL
LIN {X 0,Y 496.933,Z 725.074,A -85,B 0,C 180,E1 24044.211,E2 24044.211} C_VEL
LIN {X 0,Y 496.533,Z 736.441,A -85,B 0,C 180,E1 24042.325,E2 24042.325} C_VEL
LIN {X 0,Y 496.279,Z 746.171,A -85,B 0,C 180,E1 24040.33,E2 24040.33} C_VEL
LIN {X 0,Y 496.116,Z 754.038,A -85,B 0,C 180,E1 24038.289,E2 24038.289} C_VEL
LIN {X 0,Y 496.025,Z 760.009,A -85,B 0,C 180,E1 24036.25,E2 24036.25} C_VEL
LIN {X 0,Y 495.993,Z 764.303,A -85,B 0,C 180,E1 24034.163,E2 24034.163} C_VEL
LIN {X 0,Y 495.99,Z 766.848,A -85,B 0,C 180,E1 24032.08,E2 24032.08} C_VEL
LIN {X 0,Y 495.995,Z 767.705,A -85,B 0,C 180,E1 24030.001,E2 24030.001} C_VEL
LIN {X 0,Y 495.986,Z 766.789,A -85,B 0,C 180,E1 24027.806,E2 24027.806} C_VEL
LIN {X 0,Y 495.982,Z 764.198,A -85,B 0,C 180,E1 24025.723,E2 24025.723} C_VEL
LIN {X 0,Y 496.011,Z 759.813,A -85,B 0,C 180,E1 24023.614,E2 24023.614} C_VEL
LIN {X 0,Y 496.108,Z 753.685,A -85,B 0,C 180,E1 24021.541,E2 24021.541} C_VEL
LIN {X 0,Y 496.279,Z 745.652,A -85,B 0,C 180,E1 24019.478,E2 24019.478} C_VEL
LIN {X 0,Y 496.543,Z 736.259,A -85,B 0,C 180,E1 24017.558,E2 24017.558} C_VEL
LIN {X 0,Y 496.963,Z 724.933,A -85,B 0,C 180,E1 24015.673,E2 24015.673} C_VEL
LIN {X 0,Y 497.453,Z 712.971,A -85,B 0,C 180,E1 24014.017,E2 24014.017} C_VEL
LIN {X 0,Y 498.096,Z 699.122,A -85,B 0,C 180,E1 24012.417,E2 24012.417} C_VEL
LIN {X 0,Y 498.793,Z 684.332,A -85,B 0,C 180,E1 24010.991,E2 24010.991} C_VEL
LIN {X 0,Y 499.524,Z 668.726,A -85,B 0,C 180,E1 24009.741,E2 24009.741} C_VEL
LIN {X 0,Y 500.288,Z 651.973,A -85,B 0,C 180,E1 24008.645,E2 24008.645} C_VEL
LIN {X 0,Y 501.02,Z 634.195,A -85,B 0,C 180,E1 24007.719,E2 24007.719} C_VEL
LIN {X 0,Y 501.677,Z 615.492,A -85,B 0,C 180,E1 24006.98,E2 24006.98} C_VEL
LIN {X 0,Y 502.21,Z 596.326,A -85,B 0,C 180,E1 24006.452,E2 24006.452} C_VEL
LIN {X 0,Y 502.556,Z 567.237,A -85,B 0,C 180,E1 24005.976,E2 24005.976} C_VEL
LIN {X 0,Y 503.982,Z 400.206,A -85,B 0,C 180,E1 24003.461,E2 24003.461} C_VEL
LIN {X 0,Y 502.29,Z 386.891,A -85,B 0,C 180,E1 24003.138,E2 24003.138} C_VEL
LIN {X 0,Y 504.291,Z 342.462,A -85,B 0,C 180,E1 23999.556,E2 23999.556} C_VEL
LIN {X 0,Y 505.663,Z 314.767,A -85,B 0,C 180,E1 23997.257,E2 23997.257} C_VEL
LIN {X 0,Y 498.472,Z 294.27,A -85,B 0,C 180,E1 23994.925,E2 23994.925} C_VEL
LIN {X 0,Y 496.71,Z 288.928,A -85,B 0,C 180,E1 23994.286,E2 23994.286} C_VEL
LIN {X 0,Y 496.689,Z 288.926,A -85,B 0,C 180,E1 23990.808,E2 23990.808} C_VEL
LIN {X 0,Y 496.724,Z 288.924,A -85,B 0,C 180,E1 23987.443,E2 23987.443} C_VEL
LIN {X 0,Y 496.732,Z 288.924,A -85,B 0,C 180,E1 23983.984,E2 23983.984} C_VEL
LIN {X 0,Y 496.69,Z 288.925,A -85,B 0,C 180,E1 23980.559,E2 23980.559} C_VEL
LIN {X 0,Y 496.693,Z 288.922,A -85,B 0,C 180,E1 23976.951,E2 23976.951} C_VEL
LIN {X 0,Y 496.746,Z 288.922,A -85,B 0,C 180,E1 23973.562,E2 23973.562} C_VEL
LIN {X 0,Y 496.709,Z 288.922,A -85,B 0,C 180,E1 23970.216,E2 23970.216} C_VEL
LIN {X 0,Y 496.693,Z 288.922,A -85,B 0,C 180,E1 23966.804,E2 23966.804} C_VEL
LIN {X 0,Y 496.731,Z 288.921,A -85,B 0,C 180,E1 23963.363,E2 23963.363} C_VEL
LIN {X 0,Y 496.732,Z 288.922,A -85,B 0,C 180,E1 23959.95,E2 23959.95} C_VEL
LIN {X 0,Y 496.696,Z 288.922,A -85,B 0,C 180,E1 23956.611,E2 23956.611} C_VEL
LIN {X 0,Y 496.716,Z 288.921,A -85,B 0,C 180,E1 23953.149,E2 23953.149} C_VEL
LIN {X 0,Y 496.751,Z 288.923,A -85,B 0,C 180,E1 23949.735,E2 23949.735} C_VEL
LIN {X 0,Y 496.701,Z 288.922,A -85,B 0,C 180,E1 23946.358,E2 23946.358} C_VEL
LIN {X 0,Y 496.701,Z 288.921,A -85,B 0,C 180,E1 23942.771,E2 23942.771} C_VEL
LIN {X 0,Y 496.756,Z 288.92,A -85,B 0,C 180,E1 23939.425,E2 23939.425} C_VEL
LIN {X 0,Y 496.728,Z 288.922,A -85,B 0,C 180,E1 23935.962,E2 23935.962} C_VEL
LIN {X 0,Y 496.703,Z 288.921,A -85,B 0,C 180,E1 23932.6,E2 23932.6} C_VEL
LIN {X 0,Y 496.736,Z 288.92,A -85,B 0,C 180,E1 23929.19,E2 23929.19} C_VEL
LIN {X 0,Y 496.743,Z 288.922,A -85,B 0,C 180,E1 23925.787,E2 23925.787} C_VEL
LIN {X 0,Y 496.705,Z 288.921,A -85,B 0,C 180,E1 23922.428,E2 23922.428} C_VEL
LIN {X 0,Y 496.727,Z 288.919,A -85,B 0,C 180,E1 23919.007,E2 23919.007} C_VEL
LIN {X 0,Y 496.755,Z 288.923,A -85,B 0,C 180,E1 23915.633,E2 23915.633} C_VEL
LIN {X 0,Y 496.716,Z 288.921,A -85,B 0,C 180,E1 23912.163,E2 23912.163} C_VEL
LIN {X 0,Y 496.71,Z 288.92,A -85,B 0,C 180,E1 23908.579,E2 23908.579} C_VEL
LIN {X 0,Y 496.746,Z 288.919,A -85,B 0,C 180,E1 23905.138,E2 23905.138} C_VEL
LIN {X 0,Y 496.749,Z 288.922,A -85,B 0,C 180,E1 23901.691,E2 23901.691} C_VEL
LIN {X 0,Y 496.713,Z 288.92,A -85,B 0,C 180,E1 23898.313,E2 23898.313} C_VEL
LIN {X 0,Y 496.721,Z 288.919,A -85,B 0,C 180,E1 23894.723,E2 23894.723} C_VEL
LIN {X 0,Y 496.771,Z 288.918,A -85,B 0,C 180,E1 23891.311,E2 23891.311} C_VEL
LIN {X 0,Y 496.73,Z 288.921,A -85,B 0,C 180,E1 23887.873,E2 23887.873} C_VEL
LIN {X 0,Y 496.715,Z 288.92,A -85,B 0,C 180,E1 23886.215,E2 23886.215} C_VEL
LIN {X 0,Y 495.737,Z 289.047,A -85,B 0,C 180,E1 23885.326,E2 23885.326} C_VEL
LIN {X 0,Y 489.211,Z 289.856,A -85,B 0,C 180,E1 23882.763,E2 23882.763} C_VEL
LIN {X 0,Y 488.779,Z 289.909,A -85,B 0,C 180,E1 23882.176,E2 23882.176} C_VEL
LIN {X 0,Y 488.783,Z 289.907,A -85,B 0,C 180,E1 23878.598,E2 23878.598} C_VEL
LIN {X 0,Y 488.826,Z 289.907,A -85,B 0,C 180,E1 23875.178,E2 23875.178} C_VEL
LIN {X 0,Y 488.801,Z 289.91,A -85,B 0,C 180,E1 23871.729,E2 23871.729} C_VEL
LIN {X 0,Y 488.78,Z 289.908,A -85,B 0,C 180,E1 23868.238,E2 23868.238} C_VEL
LIN {X 0,Y 488.793,Z 289.907,A -85,B 0,C 180,E1 23864.693,E2 23864.693} C_VEL
LIN {X 0,Y 488.832,Z 289.907,A -85,B 0,C 180,E1 23861.204,E2 23861.204} C_VEL
LIN {X 0,Y 488.808,Z 289.91,A -85,B 0,C 180,E1 23857.64,E2 23857.64} C_VEL
LIN {X 0,Y 488.781,Z 289.908,A -85,B 0,C 180,E1 23854.222,E2 23854.222} C_VEL
LIN {X 0,Y 488.802,Z 289.906,A -85,B 0,C 180,E1 23850.702,E2 23850.702} C_VEL
LIN {X 0,Y 488.832,Z 289.907,A -85,B 0,C 180,E1 23847.185,E2 23847.185} C_VEL
LIN {X 0,Y 488.805,Z 289.91,A -85,B 0,C 180,E1 23843.657,E2 23843.657} C_VEL
LIN {X 0,Y 488.785,Z 289.907,A -85,B 0,C 180,E1 23840.224,E2 23840.224} C_VEL
LIN {X 0,Y 488.813,Z 289.905,A -85,B 0,C 180,E1 23836.755,E2 23836.755} C_VEL
LIN {X 0,Y 488.831,Z 289.908,A -85,B 0,C 180,E1 23833.237,E2 23833.237} C_VEL
LIN {X 0,Y 488.797,Z 289.909,A -85,B 0,C 180,E1 23829.775,E2 23829.775} C_VEL
LIN {X 0,Y 488.791,Z 289.906,A -85,B 0,C 180,E1 23826.235,E2 23826.235} C_VEL
LIN {X 0,Y 488.82,Z 289.904,A -85,B 0,C 180,E1 23822.729,E2 23822.729} C_VEL
LIN {X 0,Y 488.836,Z 289.908,A -85,B 0,C 180,E1 23819.206,E2 23819.206} C_VEL
LIN {X 0,Y 488.806,Z 289.909,A -85,B 0,C 180,E1 23815.627,E2 23815.627} C_VEL
LIN {X 0,Y 488.794,Z 289.906,A -85,B 0,C 180,E1 23812.143,E2 23812.143} C_VEL
LIN {X 0,Y 488.82,Z 289.904,A -85,B 0,C 180,E1 23808.645,E2 23808.645} C_VEL
LIN {X 0,Y 488.833,Z 289.909,A -85,B 0,C 180,E1 23805.045,E2 23805.045} C_VEL
LIN {X 0,Y 488.812,Z 289.909,A -85,B 0,C 180,E1 23801.506,E2 23801.506} C_VEL
LIN {X 0,Y 488.795,Z 289.909,A -85,B 0,C 180,E1 23798.001,E2 23798.001} C_VEL
LIN {X 0,Y 488.814,Z 289.908,A -85,B 0,C 180,E1 23794.478,E2 23794.478} C_VEL
LIN {X 0,Y 488.855,Z 290.154,A -85,B 0,C 180,E1 23791.365,E2 23791.365} C_VEL
LIN {X 0,Y 493.858,Z 309.006,A -85,B 0,C 180,E1 23788.516,E2 23788.516} C_VEL
LIN {X 0,Y 494.095,Z 312.83,A -85,B 0,C 180,E1 23787.998,E2 23787.998} C_VEL
LIN {X 0,Y 492.752,Z 341.722,A -85,B 0,C 180,E1 23784.323,E2 23784.323} C_VEL
LIN {X 0,Y 491.531,Z 371.411,A -85,B 0,C 180,E1 23780.602,E2 23780.602} C_VEL
LIN {X 0,Y 490.455,Z 400.325,A -85,B 0,C 180,E1 23777.034,E2 23777.034} C_VEL
LIN {X 0,Y 490.424,Z 404.228,A -85,B 0,C 180,E1 23776.596,E2 23776.596} C_VEL
LIN {X 0,Y 492.402,Z 418.347,A -85,B 0,C 180,E1 23776.271,E2 23776.271} C_VEL
LIN {X 0,Y 491.204,Z 521.069,A -85,B 0,C 180,E1 23774.546,E2 23774.546} C_VEL
LIN {X 0,Y 490.952,Z 536.096,A -85,B 0,C 180,E1 23774.084,E2 23774.084} C_VEL
LIN {X 0,Y 490.583,Z 551.375,A -85,B 0,C 180,E1 23773.373,E2 23773.373} C_VEL
LIN {X 0,Y 490.141,Z 566.033,A -85,B 0,C 180,E1 23772.426,E2 23772.426} C_VEL
LIN {X 0,Y 489.727,Z 578.569,A -85,B 0,C 180,E1 23771.361,E2 23771.361} C_VEL
LIN {X 0,Y 489.368,Z 589.103,A -85,B 0,C 180,E1 23770.237,E2 23770.237} C_VEL
LIN {X 0,Y 489.005,Z 599.564,A -85,B 0,C 180,E1 23768.819,E2 23768.819} C_VEL
LIN {X 0,Y 488.745,Z 607.734,A -85,B 0,C 180,E1 23767.403,E2 23767.403} C_VEL
LIN {X 0,Y 488.572,Z 614.58,A -85,B 0,C 180,E1 23765.871,E2 23765.871} C_VEL
LIN {X 0,Y 488.456,Z 619.918,A -85,B 0,C 180,E1 23764.224,E2 23764.224} C_VEL
LIN {X 0,Y 488.403,Z 623.508,A -85,B 0,C 180,E1 23762.58,E2 23762.58} C_VEL
LIN {X 0,Y 488.4,Z 625.566,A -85,B 0,C 180,E1 23760.702,E2 23760.702} C_VEL
LIN {X 0,Y 488.424,Z 625.59,A -85,B 0,C 180,E1 23758.943,E2 23758.943} C_VEL
LIN {X 0,Y 488.485,Z 623.977,A -85,B 0,C 180,E1 23757.283,E2 23757.283} C_VEL
LIN {X 0,Y 488.599,Z 620.425,A -85,B 0,C 180,E1 23755.538,E2 23755.538} C_VEL
LIN {X 0,Y 488.762,Z 615.213,A -85,B 0,C 180,E1 23753.892,E2 23753.892} C_VEL
LIN {X 0,Y 488.996,Z 608.553,A -85,B 0,C 180,E1 23752.361,E2 23752.361} C_VEL
LIN {X 0,Y 489.327,Z 599.683,A -85,B 0,C 180,E1 23750.828,E2 23750.828} C_VEL
LIN {X 0,Y 489.724,Z 589.54,A -85,B 0,C 180,E1 23749.47,E2 23749.47} C_VEL
LIN {X 0,Y 490.137,Z 578.398,A -85,B 0,C 180,E1 23748.291,E2 23748.291} C_VEL
LIN {X 0,Y 490.629,Z 564.632,A -85,B 0,C 180,E1 23747.164,E2 23747.164} C_VEL
LIN {X 0,Y 491.056,Z 550.228,A -85,B 0,C 180,E1 23746.277,E2 23746.277} C_VEL
LIN {X 0,Y 491.414,Z 535.503,A -85,B 0,C 180,E1 23745.618,E2 23745.618} C_VEL
LIN {X 0,Y 491.669,Z 520.209,A -85,B 0,C 180,E1 23745.159,E2 23745.159} C_VEL
LIN {X 0,Y 494.015,Z 418.006,A -85,B 0,C 180,E1 23743.141,E2 23743.141} C_VEL
LIN {X 0,Y 491.474,Z 403.826,A -85,B 0,C 180,E1 23742.659,E2 23742.659} C_VEL
LIN {X 0,Y 492.944,Z 373.894,A -85,B 0,C 180,E1 23738.834,E2 23738.834} C_VEL
LIN {X 0,Y 494.666,Z 346.653,A -85,B 0,C 180,E1 23735.265,E2 23735.265} C_VEL
LIN {X 0,Y 496.711,Z 320.432,A -85,B 0,C 180,E1 23731.701,E2 23731.701} C_VEL
LIN {X 0,Y 497.042,Z 315.872,A -85,B 0,C 180,E1 23731.053,E2 23731.053} C_VEL
LIN {X 0,Y 493.936,Z 304.592,A -85,B 0,C 180,E1 23728.983,E2 23728.983} C_VEL
LIN {X 0,Y 491.015,Z 296.087,A -85,B 0,C 180,E1 23727.202,E2 23727.202} C_VEL
LIN {X 0,Y 488.808,Z 289.912,A -85,B 0,C 180,E1 23725.73,E2 23725.73} C_VEL
LIN {X 0,Y 488.827,Z 289.908,A -85,B 0,C 180,E1 23722.143,E2 23722.143} C_VEL
LIN {X 0,Y 488.82,Z 289.91,A -85,B 0,C 180,E1 23718.647,E2 23718.647} C_VEL
LIN {X 0,Y 488.81,Z 289.911,A -85,B 0,C 180,E1 23715.052,E2 23715.052} C_VEL
LIN {X 0,Y 488.82,Z 289.911,A -85,B 0,C 180,E1 23711.509,E2 23711.509} C_VEL
LIN {X 0,Y 488.836,Z 289.909,A -85,B 0,C 180,E1 23708.001,E2 23708.001} C_VEL
LIN {X 0,Y 488.841,Z 290.034,A -85,B 0,C 180,E1 23707.778,E2 23707.778} C_VEL
LIN {X 0,Y 490.148,Z 293.482,A -85,B 0,C 180,E1 23707.097,E2 23707.097} C_VEL
LIN {X 0,Y 493.447,Z 301.417,A -85,B 0,C 180,E1 23705.655,E2 23705.655} C_VEL
LIN {X 0,Y 497.214,Z 311.834,A -85,B 0,C 180,E1 23704.054,E2 23704.054} C_VEL
LIN {X 0,Y 499.281,Z 318.574,A -85,B 0,C 180,E1 23703.142,E2 23703.142} C_VEL
LIN {X 0,Y 496.598,Z 351.395,A -85,B 0,C 180,E1 23700.156,E2 23700.156} C_VEL
LIN {X 0,Y 494.495,Z 388.898,A -85,B 0,C 180,E1 23696.99,E2 23696.99} C_VEL
LIN {X 0,Y 496.121,Z 403.915,A -85,B 0,C 180,E1 23696.655,E2 23696.655} C_VEL
LIN {X 0,Y 494.615,Z 547.012,A -85,B 0,C 180,E1 23694.433,E2 23694.433} C_VEL
LIN {X 0,Y 494.185,Z 592.847,A -85,B 0,C 180,E1 23693.727,E2 23693.727} C_VEL
LIN {X 0,Y 493.663,Z 611.78,A -85,B 0,C 180,E1 23693.228,E2 23693.228} C_VEL
LIN {X 0,Y 493.037,Z 630.645,A -85,B 0,C 180,E1 23692.507,E2 23692.507} C_VEL
LIN {X 0,Y 492.309,Z 649.066,A -85,B 0,C 180,E1 23691.569,E2 23691.569} C_VEL
LIN {X 0,Y 491.554,Z 665.968,A -85,B 0,C 180,E1 23690.48,E2 23690.48} C_VEL
LIN {X 0,Y 490.813,Z 682.034,A -85,B 0,C 180,E1 23689.209,E2 23689.209} C_VEL
LIN {X 0,Y 490.118,Z 697.191,A -85,B 0,C 180,E1 23687.758,E2 23687.758} C_VEL
LIN {X 0,Y 489.479,Z 711.332,A -85,B 0,C 180,E1 23686.13,E2 23686.13} C_VEL
LIN {X 0,Y 488.961,Z 724.315,A -85,B 0,C 180,E1 23684.326,E2 23684.326} C_VEL
LIN {X 0,Y 488.554,Z 735.624,A -85,B 0,C 180,E1 23682.41,E2 23682.41} C_VEL
LIN {X 0,Y 488.314,Z 744.828,A -85,B 0,C 180,E1 23680.501,E2 23680.501} C_VEL
LIN {X 0,Y 488.161,Z 752.587,A -85,B 0,C 180,E1 23678.481,E2 23678.481} C_VEL
LIN {X 0,Y 488.075,Z 758.52,A -85,B 0,C 180,E1 23676.47,E2 23676.47} C_VEL
LIN {X 0,Y 488.056,Z 762.959,A -85,B 0,C 180,E1 23674.348,E2 23674.348} C_VEL
LIN {X 0,Y 488.064,Z 765.622,A -85,B 0,C 180,E1 23672.232,E2 23672.232} C_VEL
LIN {X 0,Y 488.071,Z 766.572,A -85,B 0,C 180,E1 23670.118,E2 23670.118} C_VEL
LIN {X 0,Y 488.061,Z 765.842,A -85,B 0,C 180,E1 23668.005,E2 23668.005} C_VEL
LIN {X 0,Y 488.049,Z 763.428,A -85,B 0,C 180,E1 23665.889,E2 23665.889} C_VEL
LIN {X 0,Y 488.061,Z 759.278,A -85,B 0,C 180,E1 23663.768,E2 23663.768} C_VEL
LIN {X 0,Y 488.129,Z 753.656,A -85,B 0,C 180,E1 23661.757,E2 23661.757} C_VEL
LIN {X 0,Y 488.272,Z 746.258,A -85,B 0,C 180,E1 23659.739,E2 23659.739} C_VEL
LIN {X 0,Y 488.507,Z 737.475,A -85,B 0,C 180,E1 23657.831,E2 23657.831} C_VEL
LIN {X 0,Y 488.898,Z 726.671,A -85,B 0,C 180,E1 23655.915,E2 23655.915} C_VEL
LIN {X 0,Y 489.415,Z 714.343,A -85,B 0,C 180,E1 23654.113,E2 23654.113} C_VEL
LIN {X 0,Y 490.094,Z 700.448,A -85,B 0,C 180,E1 23652.427,E2 23652.427} C_VEL
LIN {X 0,Y 490.839,Z 685.736,A -85,B 0,C 180,E1 23650.943,E2 23650.943} C_VEL
LIN {X 0,Y 491.664,Z 669.47,A -85,B 0,C 180,E1 23649.589,E2 23649.589} C_VEL
LIN {X 0,Y 492.501,Z 652.489,A -85,B 0,C 180,E1 23648.442,E2 23648.442} C_VEL
LIN {X 0,Y 493.276,Z 635.215,A -85,B 0,C 180,E1 23647.51,E2 23647.51} C_VEL
LIN {X 0,Y 493.983,Z 616.909,A -85,B 0,C 180,E1 23646.754,E2 23646.754} C_VEL
LIN {X 0,Y 494.554,Z 598.359,A -85,B 0,C 180,E1 23646.21,E2 23646.21} C_VEL
LIN {X 0,Y 494.91,Z 576.02,A -85,B 0,C 180,E1 23645.808,E2 23645.808} C_VEL
LIN {X 0,Y 496.576,Z 401.223,A -85,B 0,C 180,E1 23643.125,E2 23643.125} C_VEL
LIN {X 0,Y 494.782,Z 387.195,A -85,B 0,C 180,E1 23642.794,E2 23642.794} C_VEL
LIN {X 0,Y 496.931,Z 343.687,A -85,B 0,C 180,E1 23639.223,E2 23639.223} C_VEL
LIN {X 0,Y 498.334,Z 317.413,A -85,B 0,C 180,E1 23637.002,E2 23637.002} C_VEL
LIN {X 0,Y 490.822,Z 295.889,A -85,B 0,C 180,E1 23634.51,E2 23634.51} C_VEL
LIN {X 0,Y 488.81,Z 289.912,A -85,B 0,C 180,E1 23633.763,E2 23633.763} C_VEL
LIN {X 0,Y 488.769,Z 289.915,A -85,B 0,C 180,E1 23630.281,E2 23630.281} C_VEL
LIN {X 0,Y 488.752,Z 289.914,A -85,B 0,C 180,E1 23626.901,E2 23626.901} C_VEL
LIN {X 0,Y 488.785,Z 289.912,A -85,B 0,C 180,E1 23623.42,E2 23623.42} C_VEL
LIN {X 0,Y 488.795,Z 289.914,A -85,B 0,C 180,E1 23619.965,E2 23619.965} C_VEL
LIN {X 0,Y 488.752,Z 289.911,A -85,B 0,C 180,E1 23616.536,E2 23616.536} C_VEL
LIN {X 0,Y 488.759,Z 289.911,A -85,B 0,C 180,E1 23612.968,E2 23612.968} C_VEL
LIN {X 0,Y 488.808,Z 289.91,A -85,B 0,C 180,E1 23609.537,E2 23609.537} C_VEL
LIN {X 0,Y 488.78,Z 289.911,A -85,B 0,C 180,E1 23606.093,E2 23606.093} C_VEL
LIN {X 0,Y 488.755,Z 289.911,A -85,B 0,C 180,E1 23602.62,E2 23602.62} C_VEL
LIN {X 0,Y 488.772,Z 289.91,A -85,B 0,C 180,E1 23599.107,E2 23599.107} C_VEL
LIN {X 0,Y 488.821,Z 289.912,A -85,B 0,C 180,E1 23595.666,E2 23595.666} C_VEL
LIN {X 0,Y 488.766,Z 289.911,A -85,B 0,C 180,E1 23592.285,E2 23592.285} C_VEL
LIN {X 0,Y 488.759,Z 289.91,A -85,B 0,C 180,E1 23588.709,E2 23588.709} C_VEL
LIN {X 0,Y 488.807,Z 289.91,A -85,B 0,C 180,E1 23585.401,E2 23585.401} C_VEL
LIN {X 0,Y 488.797,Z 289.911,A -85,B 0,C 180,E1 23581.877,E2 23581.877} C_VEL
LIN {X 0,Y 488.763,Z 289.91,A -85,B 0,C 180,E1 23578.478,E2 23578.478} C_VEL
LIN {X 0,Y 488.774,Z 289.909,A -85,B 0,C 180,E1 23574.955,E2 23574.955} C_VEL
LIN {X 0,Y 488.826,Z 289.91,A -85,B 0,C 180,E1 23571.533,E2 23571.533} C_VEL
LIN {X 0,Y 488.789,Z 289.91,A -85,B 0,C 180,E1 23567.959,E2 23567.959} C_VEL
LIN {X 0,Y 488.766,Z 289.909,A -85,B 0,C 180,E1 23564.579,E2 23564.579} C_VEL
LIN {X 0,Y 488.798,Z 289.908,A -85,B 0,C 180,E1 23561.146,E2 23561.146} C_VEL
LIN {X 0,Y 488.819,Z 289.911,A -85,B 0,C 180,E1 23557.64,E2 23557.64} C_VEL
LIN {X 0,Y 488.775,Z 289.91,A -85,B 0,C 180,E1 23554.166,E2 23554.166} C_VEL
LIN {X 0,Y 488.77,Z 289.909,A -85,B 0,C 180,E1 23550.599,E2 23550.599} C_VEL
LIN {X 0,Y 488.811,Z 289.908,A -85,B 0,C 180,E1 23547.179,E2 23547.179} C_VEL
LIN {X 0,Y 488.816,Z 289.911,A -85,B 0,C 180,E1 23543.62,E2 23543.62} C_VEL
LIN {X 0,Y 488.774,Z 289.91,A -85,B 0,C 180,E1 23540.19,E2 23540.19} C_VEL
LIN {X 0,Y 488.774,Z 289.908,A -85,B 0,C 180,E1 23536.568,E2 23536.568} C_VEL
LIN {X 0,Y 488.811,Z 289.907,A -85,B 0,C 180,E1 23533.092,E2 23533.092} C_VEL
LIN {X 0,Y 488.812,Z 289.91,A -85,B 0,C 180,E1 23529.656,E2 23529.656} C_VEL
LIN {X 0,Y 488.777,Z 289.909,A -85,B 0,C 180,E1 23526.213,E2 23526.213} C_VEL
LIN {X 0,Y 488.781,Z 289.908,A -85,B 0,C 180,E1 23522.569,E2 23522.569} C_VEL
LIN {X 0,Y 488.779,Z 289.909,A -85,B 0,C 180,E1 23522.176,E2 23522.176} C_VEL
LIN {X 0,Y 487.796,Z 290.036,A -85,B 0,C 180,E1 23521.272,E2 23521.272} C_VEL
LIN {X 0,Y 481.268,Z 290.845,A -85,B 0,C 180,E1 23518.667,E2 23518.667} C_VEL
LIN {X 0,Y 480.844,Z 290.898,A -85,B 0,C 180,E1 23518.07,E2 23518.07} C_VEL
LIN {X 0,Y 480.842,Z 290.897,A -85,B 0,C 180,E1 23514.443,E2 23514.443} C_VEL
LIN {X 0,Y 480.874,Z 290.895,A -85,B 0,C 180,E1 23510.954,E2 23510.954} C_VEL
LIN {X 0,Y 480.889,Z 290.899,A -85,B 0,C 180,E1 23507.389,E2 23507.389} C_VEL
LIN {X 0,Y 480.849,Z 290.898,A -85,B 0,C 180,E1 23503.957,E2 23503.957} C_VEL
LIN {X 0,Y 480.845,Z 290.896,A -85,B 0,C 180,E1 23500.422,E2 23500.422} C_VEL
LIN {X 0,Y 480.879,Z 290.894,A -85,B 0,C 180,E1 23496.926,E2 23496.926} C_VEL
LIN {X 0,Y 480.888,Z 290.899,A -85,B 0,C 180,E1 23493.337,E2 23493.337} C_VEL
LIN {X 0,Y 480.852,Z 290.898,A -85,B 0,C 180,E1 23489.88,E2 23489.88} C_VEL
LIN {X 0,Y 480.847,Z 290.896,A -85,B 0,C 180,E1 23486.303,E2 23486.303} C_VEL
LIN {X 0,Y 480.878,Z 290.894,A -85,B 0,C 180,E1 23482.833,E2 23482.833} C_VEL
LIN {X 0,Y 480.892,Z 290.897,A -85,B 0,C 180,E1 23479.214,E2 23479.214} C_VEL
LIN {X 0,Y 480.864,Z 290.898,A -85,B 0,C 180,E1 23475.673,E2 23475.673} C_VEL
LIN {X 0,Y 480.849,Z 290.896,A -85,B 0,C 180,E1 23472.201,E2 23472.201} C_VEL
LIN {X 0,Y 480.87,Z 290.894,A -85,B 0,C 180,E1 23468.661,E2 23468.661} C_VEL
LIN {X 0,Y 480.894,Z 290.896,A -85,B 0,C 180,E1 23465.165,E2 23465.165} C_VEL
LIN {X 0,Y 480.872,Z 290.898,A -85,B 0,C 180,E1 23461.565,E2 23461.565} C_VEL
LIN {X 0,Y 480.853,Z 290.896,A -85,B 0,C 180,E1 23458.03,E2 23458.03} C_VEL
LIN {X 0,Y 480.861,Z 290.894,A -85,B 0,C 180,E1 23454.386,E2 23454.386} C_VEL
LIN {X 0,Y 480.894,Z 290.892,A -85,B 0,C 180,E1 23450.796,E2 23450.796} C_VEL
LIN {X 0,Y 480.892,Z 290.897,A -85,B 0,C 180,E1 23447.164,E2 23447.164} C_VEL
LIN {X 0,Y 480.865,Z 290.897,A -85,B 0,C 180,E1 23443.647,E2 23443.647} C_VEL
LIN {X 0,Y 480.857,Z 290.898,A -85,B 0,C 180,E1 23440.075,E2 23440.075} C_VEL
LIN {X 0,Y 480.884,Z 290.896,A -85,B 0,C 180,E1 23436.622,E2 23436.622} C_VEL
LIN {X 0,Y 480.895,Z 290.896,A -85,B 0,C 180,E1 23433.004,E2 23433.004} C_VEL
LIN {X 0,Y 480.868,Z 290.973,A -85,B 0,C 180,E1 23431.807,E2 23431.807} C_VEL
LIN {X 0,Y 486.138,Z 310.763,A -85,B 0,C 180,E1 23428.766,E2 23428.766} C_VEL
LIN {X 0,Y 486.585,Z 313.784,A -85,B 0,C 180,E1 23428.335,E2 23428.335} C_VEL
LIN {X 0,Y 485.15,Z 342.367,A -85,B 0,C 180,E1 23424.649,E2 23424.649} C_VEL
LIN {X 0,Y 483.864,Z 371.706,A -85,B 0,C 180,E1 23420.929,E2 23420.929} C_VEL
LIN {X 0,Y 482.708,Z 400.276,A -85,B 0,C 180,E1 23417.352,E2 23417.352} C_VEL
LIN {X 0,Y 482.658,Z 404.09,A -85,B 0,C 180,E1 23416.919,E2 23416.919} C_VEL
LIN {X 0,Y 484.805,Z 419.205,A -85,B 0,C 180,E1 23416.557,E2 23416.557} C_VEL
LIN {X 0,Y 483.484,Z 521.734,A -85,B 0,C 180,E1 23414.784,E2 23414.784} C_VEL
LIN {X 0,Y 483.216,Z 536.684,A -85,B 0,C 180,E1 23414.314,E2 23414.314} C_VEL
LIN {X 0,Y 482.833,Z 551.697,A -85,B 0,C 180,E1 23413.607,E2 23413.607} C_VEL
LIN {X 0,Y 482.384,Z 565.867,A -85,B 0,C 180,E1 23412.69,E2 23412.69} C_VEL
LIN {X 0,Y 481.96,Z 578.056,A -85,B 0,C 180,E1 23411.668,E2 23411.668} C_VEL
LIN {X 0,Y 481.533,Z 589.901,A -85,B 0,C 180,E1 23410.406,E2 23410.406} C_VEL
LIN {X 0,Y 481.142,Z 600.43,A -85,B 0,C 180,E1 23408.965,E2 23408.965} C_VEL
LIN {X 0,Y 480.863,Z 608.674,A -85,B 0,C 180,E1 23407.525,E2 23407.525} C_VEL
LIN {X 0,Y 480.673,Z 615.58,A -85,B 0,C 180,E1 23405.968,E2 23405.968} C_VEL
LIN {X 0,Y 480.545,Z 620.975,A -85,B 0,C 180,E1 23404.294,E2 23404.294} C_VEL
LIN {X 0,Y 480.488,Z 624.618,A -85,B 0,C 180,E1 23402.622,E2 23402.622} C_VEL
LIN {X 0,Y 480.485,Z 626.726,A -85,B 0,C 180,E1 23400.714,E2 23400.714} C_VEL
LIN {X 0,Y 480.515,Z 626.781,A -85,B 0,C 180,E1 23398.925,E2 23398.925} C_VEL
LIN {X 0,Y 480.587,Z 625.224,A -85,B 0,C 180,E1 23397.256,E2 23397.256} C_VEL
LIN {X 0,Y 480.717,Z 621.655,A -85,B 0,C 180,E1 23395.465,E2 23395.465} C_VEL
LIN {X 0,Y 480.9,Z 616.443,A -85,B 0,C 180,E1 23393.792,E2 23393.792} C_VEL
LIN {X 0,Y 481.161,Z 609.776,A -85,B 0,C 180,E1 23392.236,E2 23392.236} C_VEL
LIN {X 0,Y 481.521,Z 600.892,A -85,B 0,C 180,E1 23390.678,E2 23390.678} C_VEL
LIN {X 0,Y 481.955,Z 590.775,A -85,B 0,C 180,E1 23389.298,E2 23389.298} C_VEL
LIN {X 0,Y 482.409,Z 579.665,A -85,B 0,C 180,E1 23388.097,E2 23388.097} C_VEL
LIN {X 0,Y 482.938,Z 566.049,A -85,B 0,C 180,E1 23386.956,E2 23386.956} C_VEL
LIN {X 0,Y 483.398,Z 551.821,A -85,B 0,C 180,E1 23386.055,E2 23386.055} C_VEL
LIN {X 0,Y 483.775,Z 537.667,A -85,B 0,C 180,E1 23385.394,E2 23385.394} C_VEL
LIN {X 0,Y 484.073,Z 521.983,A -85,B 0,C 180,E1 23384.894,E2 23384.894} C_VEL
LIN {X 0,Y 486.613,Z 418.259,A -85,B 0,C 180,E1 23382.736,E2 23382.736} C_VEL
LIN {X 0,Y 483.989,Z 403.643,A -85,B 0,C 180,E1 23382.195,E2 23382.195} C_VEL
